ABB RobotStudio station: AutoDataCollectionRBSDone.rspag

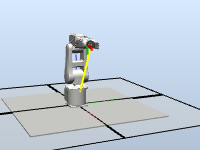
--- station ---
Station Project1 (saved by RobotStudio 6.5.7558.2005)
Controller 120-501447, task T_ROB1: task frame (RAPID world) sits at (0, 0, 10) mm in the station
Controller 120-501447
  mechanical unit ROB_1: IRB120_3_58__01, 6 joints, base frame (0, 0, 0) mm
Layout (positions relative to the parent item):
  - IRB120_3_58__01 [mechanism, from Robots\IRB120_3_58_G_01.rslib] at (0, 0, 10) mm; joint values [0, 0, 0, 0, 0, 0] (rad or m)
  - Table [part] at (-574.68, -626.92, 0) mm
  - tGripper [mechanism] at (374, 0, 640) mm, rotated rx 90 ry 0 rz 90 deg
      TCP tGripper at (14.1, 9.97, 139.57) mm
      links: ABB-TOOL-GRIPPER
  - Frame_1 [frame] at (14.1, -0.53, 139.57) mm
  - TestCyl [frame] at (160.39, -370.36, 110.04) mm
  - TestPap [frame] at (297.7, -422.52, 10) mm
  - Pointer [frame] at (82.12, -626.92, 10) mm
  - DegreeCheck1 [frame] at (285, -62, 10) mm
  - DegreeCheck2 [frame] at (285, 62, 10) mm
Attachment: IRB120_3_58__01 is attached to Table
Attachment: tGripper is attached to IRB120_3_58__01 / Link6
Collision set CollisionSet_2: Link1, Link2, Link3, Link4, Link5, Link6 against Table, near miss 0 m
Collision set CollisionSet_3: tGripper against Table, near miss 0 m

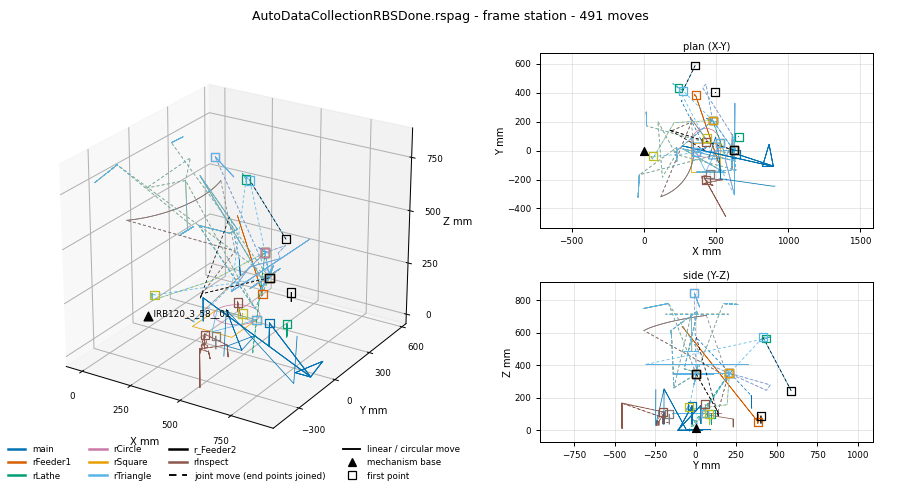
[picture p0: tool path of AutoDataCollectionRBSDone.rspag in frame station, 491 of 504 moves have a stored position in this frame; points joined in program order, loops and branches not executed]
--- Backups/120-501447/RAPID/TASK1/PROGMOD/CalibData.mod ---
MODULE CalibData
	PERS tooldata tGripper:=[TRUE,[[1.097,11.475,139.568],[0,0,0.707106781,0.707106781]],[1,[13.941,-25.105,74.149],[1,0,0,0],0,0,0]];
ENDMODULE

--- Backups/120-501447/RAPID/TASK1/PROGMOD/SERVER.mod ---
MODULE SERVER

!////////////////
!GLOBAL VARIABLES
!////////////////

!//Robot configuration
PERS tooldata currentTool := [TRUE,[[1.6,-47.2,24.1],[0.5,-0.5,-0.5,-0.5]],[1,[13.941,-25.105,74.149],[1,0,0,0],0,0,0]];
PERS wobjdata currentWobj := [FALSE,TRUE,"",[[0,0,0],[1,0,0,0]],[[0,0,0],[1,0,0,0]]];
PERS speeddata currentSpeed;
PERS zonedata currentZone;

!// Clock Synchronization
PERS bool startLog:=TRUE;
PERS bool startRob:=TRUE;

!// Mutex between logger and changing the tool and work objects
PERS bool frameMutex:=FALSE;

!//PC communication
VAR socketdev clientSocket;
VAR socketdev serverSocket;
VAR num instructionCode;
VAR num params{10};
VAR num nParams;

!PERS string ipController:= "192.168.125.1"; !robot default IP
PERS string ipController:= "127.0.0.1"; !local IP for testing in simulation
PERS num serverPort:= 5000;

!//Motion of the robot
VAR robtarget cartesianTarget;
VAR jointtarget jointsTarget;
VAR bool moveCompleted; !Set to true after finishing a Move instruction.

!//Buffered move variables
CONST num MAX_BUFFER := 512;
VAR num BUFFER_POS := 0;
VAR robtarget bufferTargets{MAX_BUFFER};
VAR speeddata bufferSpeeds{MAX_BUFFER};

!//External axis position variables
VAR extjoint externalAxis;

!//Circular move buffer
VAR robtarget circPoint;

!//Correct Instruction Execution and possible return values
VAR num ok;
CONST num SERVER_BAD_MSG :=  0;
CONST num SERVER_OK := 1;

!//Digital IO values
CONST dionum on := 1;
CONST dionum off := 0;



!////////////////
!LOCAL METHODS
!////////////////

!//Method to parse the message received from a PC
!// If correct message, loads values on:
!// - instructionCode.
!// - nParams: Number of received parameters.
!// - params{nParams}: Vector of received params.
PROC ParseMsg(string msg)
    !//Local variables
    VAR bool auxOk;
    VAR num ind:=1;
    VAR num newInd;
    VAR num length;
    VAR num indParam:=1;
    VAR string subString;
    VAR bool end := FALSE;

    !//Find the end character
    length := StrMatch(msg,1,"#");
    IF length > StrLen(msg) THEN
        !//Corrupt message
        nParams := -1;
    ELSE
        !//Read Instruction code
        newInd := StrMatch(msg,ind," ") + 1;
        subString := StrPart(msg,ind,newInd - ind - 1);
        auxOk:= StrToVal(subString, instructionCode);
        IF auxOk = FALSE THEN
            !//Impossible to read instruction code
            nParams := -1;
        ELSE
            ind := newInd;
            !//Read all instruction parameters (maximum of 8)
            WHILE end = FALSE DO
                newInd := StrMatch(msg,ind," ") + 1;
                IF newInd > length THEN
                    end := TRUE;
                ELSE
                    subString := StrPart(msg,ind,newInd - ind - 1);
                    auxOk := StrToVal(subString, params{indParam});
                    indParam := indParam + 1;
                    ind := newInd;
                ENDIF
            ENDWHILE
            nParams:= indParam - 1;
        ENDIF
    ENDIF
ENDPROC


!//Handshake between server and client:
!// - Creates socket.
!// - Waits for incoming TCP connection.
PROC ServerCreateAndConnect(string ip, num port)
    VAR string clientIP;

    SocketCreate serverSocket;
    SocketBind serverSocket, ip, port;
    SocketListen serverSocket;
    TPWrite "SERVER: Server waiting for incoming connections ...";
    WHILE SocketGetStatus(clientSocket) <> SOCKET_CONNECTED DO
        SocketAccept serverSocket,clientSocket \ClientAddress:=clientIP \Time:=WAIT_MAX;
        IF SocketGetStatus(clientSocket) <> SOCKET_CONNECTED THEN
            TPWrite "SERVER: Problem serving an incoming connection.";
            TPWrite "SERVER: Try reconnecting.";
        ENDIF
        !//Wait 0.5 seconds for the next reconnection
        WaitTime 0.5;
    ENDWHILE
    TPWrite "SERVER: Connected to IP " + clientIP;
ENDPROC


!//Parameter initialization
!// Loads default values for
!// - Tool.
!// - WorkObject.
!// - Zone.
!// - Speed.
PROC Initialize()
    currentTool := [TRUE,[[0,0,0],[1,0,0,0]],[0.001,[0,0,0.001],[1,0,0,0],0,0,0]];
    currentWobj := [FALSE,TRUE,"",[[0,0,0],[1,0,0,0]],[[0,0,0],[1,0,0,0]]];
    currentSpeed := [100, 50, 0, 0];
    currentZone := [FALSE, 0.3, 0.3,0.3,0.03,0.3,0.03]; !z0

	!Find the current external axis values so they don't move when we start
	jointsTarget := CJointT();
	externalAxis := jointsTarget.extax;
ENDPROC


!////////////////////////
!//SERVER: Main procedure
!////////////////////////
PROC main()
    !//Local variables
    VAR string receivedString;   !//Received string
    VAR string sendString;       !//Reply string
    VAR string addString;        !//String to add to the reply.
    VAR bool connected;          !//Client connected
    VAR bool reconnected;        !//Drop and reconnection happened during serving a command
    VAR robtarget cartesianPose;
    VAR jointtarget jointsPose;

    !//Motion configuration
    ConfL \Off;
    SingArea \Wrist;
    moveCompleted:= TRUE;

    !//Initialization of WorkObject, Tool, Speed and Zone
    Initialize;

    !//Socket connection
    connected:=FALSE;
    ServerCreateAndConnect ipController,serverPort;
    connected:=TRUE;

    !//Server Loop
    WHILE TRUE DO
        !//Initialization of program flow variables
        ok:=SERVER_OK;              !//Correctness of executed instruction.
        reconnected:=FALSE;         !//Has communication dropped after receiving a command?
        addString := "";

        !//Wait for a command
        SocketReceive clientSocket \Str:=receivedString \Time:=WAIT_MAX;
        ParseMsg receivedString;

        !//Execution of the command
        TEST instructionCode
            CASE 0: !Ping
                IF nParams = 0 THEN
                    ok := SERVER_OK;
                ELSE
                    ok := SERVER_BAD_MSG;
                ENDIF

            CASE 1: !Cartesian Move
                IF nParams = 7 THEN
                    cartesianTarget :=[[params{1},params{2},params{3}],
                                       [params{4},params{5},params{6},params{7}],
                                       [0,0,0,0],
                                       externalAxis];
                    ok := SERVER_OK;
                    moveCompleted := FALSE;
                    MoveL cartesianTarget, currentSpeed, currentZone, currentTool \WObj:=currentWobj ;
                    moveCompleted := TRUE;
                ELSE
                    ok := SERVER_BAD_MSG;
                ENDIF

            CASE 2: !Joint Move
                IF nParams = 6 THEN
                    jointsTarget:=[[params{1},params{2},params{3},params{4},params{5},params{6}], externalAxis];
                    ok := SERVER_OK;
                    moveCompleted := FALSE;
                    MoveAbsJ jointsTarget, currentSpeed, currentZone, currentTool \Wobj:=currentWobj;
                    moveCompleted := TRUE;
                ELSE
                    ok :=SERVER_BAD_MSG;
                ENDIF

            CASE 3: !Get Cartesian Coordinates (with current tool and workobject)
                IF nParams = 0 THEN
                    cartesianPose := CRobT(\Tool:=currentTool \WObj:=currentWObj);
                    addString := NumToStr(cartesianPose.trans.x,2) + " ";
                    addString := addString + NumToStr(cartesianPose.trans.y,2) + " ";
                    addString := addString + NumToStr(cartesianPose.trans.z,2) + " ";
                    addString := addString + NumToStr(cartesianPose.rot.q1,3) + " ";
                    addString := addString + NumToStr(cartesianPose.rot.q2,3) + " ";
                    addString := addString + NumToStr(cartesianPose.rot.q3,3) + " ";
                    addString := addString + NumToStr(cartesianPose.rot.q4,3); !End of string
                    ok := SERVER_OK;
                ELSE
                    ok :=SERVER_BAD_MSG;
                ENDIF

            CASE 4: !Get Joint Coordinates
                IF nParams = 0 THEN
                    jointsPose := CJointT();
                    addString := NumToStr(jointsPose.robax.rax_1,2) + " ";
                    addString := addString + NumToStr(jointsPose.robax.rax_2,2) + " ";
                    addString := addString + NumToStr(jointsPose.robax.rax_3,2) + " ";
                    addString := addString + NumToStr(jointsPose.robax.rax_4,2) + " ";
                    addString := addString + NumToStr(jointsPose.robax.rax_5,2) + " ";
                    addString := addString + NumToStr(jointsPose.robax.rax_6,2); !End of string
                    ok := SERVER_OK;
                ELSE
                    ok:=SERVER_BAD_MSG;
                ENDIF
			CASE 5: !Get external axis positions
                IF nParams = 0 THEN
                    jointsPose := CJointT();
                    addString := StrPart(NumToStr(jointsTarget.extax.eax_a, 2),1,8) + " ";
                    addString := addString + StrPart(NumToStr(jointsTarget.extax.eax_b,2),1,8) + " ";
                    addString := addString + StrPart(NumToStr(jointsTarget.extax.eax_c,2),1,8) + " ";
                    addString := addString + StrPart(NumToStr(jointsTarget.extax.eax_d,2),1,8) + " ";
                    addString := addString + StrPart(NumToStr(jointsTarget.extax.eax_e,2),1,8) + " ";
                    addString := addString + StrPart(NumToStr(jointsTarget.extax.eax_f,2),1,8); !End of string
                    ok := SERVER_OK;
                ELSE
                    ok:=SERVER_BAD_MSG;
                ENDIF

            CASE 6: !Set Tool
                IF nParams = 7 THEN
		   WHILE (frameMutex) DO
		        WaitTime .01; !// If the frame is being used by logger, wait here
		   ENDWHILE
		frameMutex:= TRUE;
                    currentTool.tframe.trans.x:=params{1};
                    currentTool.tframe.trans.y:=params{2};
                    currentTool.tframe.trans.z:=params{3};
                    currentTool.tframe.rot.q1:=params{4};
                    currentTool.tframe.rot.q2:=params{5};
                    currentTool.tframe.rot.q3:=params{6};
                    currentTool.tframe.rot.q4:=params{7};
                    ok := SERVER_OK;
		    frameMutex:= FALSE;
                ELSE
                    ok:=SERVER_BAD_MSG;
                ENDIF

            CASE 7: !Set Work Object
                IF nParams = 7 THEN
                    currentWobj.oframe.trans.x:=params{1};
                    currentWobj.oframe.trans.y:=params{2};
                    currentWobj.oframe.trans.z:=params{3};
                    currentWobj.oframe.rot.q1:=params{4};
                    currentWobj.oframe.rot.q2:=params{5};
                    currentWobj.oframe.rot.q3:=params{6};
                    currentWobj.oframe.rot.q4:=params{7};
                    ok := SERVER_OK;
                ELSE
                    ok:=SERVER_BAD_MSG;
                ENDIF

            CASE 8: !Set Speed of the Robot
                IF nParams = 4 THEN
                    currentSpeed.v_tcp:=params{1};
                    currentSpeed.v_ori:=params{2};
                    currentSpeed.v_leax:=params{3};
                    currentSpeed.v_reax:=params{4};
                    ok := SERVER_OK;
                ELSEIF nParams = 2 THEN
					currentSpeed.v_tcp:=params{1};
					currentSpeed.v_ori:=params{2};
					ok := SERVER_OK;
				ELSE
                    ok:=SERVER_BAD_MSG;
                ENDIF

            CASE 9: !Set zone data
                IF nParams = 4 THEN
                    IF params{1}=1 THEN
                        currentZone.finep := TRUE;
                        currentZone.pzone_tcp := 0.0;
                        currentZone.pzone_ori := 0.0;
                        currentZone.zone_ori := 0.0;
                    ELSE
                        currentZone.finep := FALSE;
                        currentZone.pzone_tcp := params{2};
                        currentZone.pzone_ori := params{3};
                        currentZone.zone_ori := params{4};
                    ENDIF
                    ok := SERVER_OK;
                ELSE
                    ok:=SERVER_BAD_MSG;
                ENDIF

            CASE 30: !Add Cartesian Coordinates to buffer
                IF nParams = 7 THEN
                    cartesianTarget :=[[params{1},params{2},params{3}],
                                        [params{4},params{5},params{6},params{7}],
                                        [0,0,0,0],
                                        externalAxis];
                    IF BUFFER_POS < MAX_BUFFER THEN
                        BUFFER_POS := BUFFER_POS + 1;
                        bufferTargets{BUFFER_POS} := cartesianTarget;
                        bufferSpeeds{BUFFER_POS} := currentSpeed;
                    ENDIF
                    ok := SERVER_OK;
                ELSE
                    ok:=SERVER_BAD_MSG;
                ENDIF

            CASE 31: !Clear Cartesian Buffer
                IF nParams = 0 THEN
                    BUFFER_POS := 0;
                    ok := SERVER_OK;
                ELSE
                    ok:=SERVER_BAD_MSG;
                ENDIF

            CASE 32: !Get Buffer Size)
                IF nParams = 0 THEN
                    addString := NumToStr(BUFFER_POS,2);
                    ok := SERVER_OK;
                ELSE
                    ok:=SERVER_BAD_MSG;
                ENDIF

            CASE 33: !Execute moves in cartesianBuffer as linear moves
                IF nParams = 0 THEN
                    FOR i FROM 1 TO (BUFFER_POS) DO
                        MoveL bufferTargets{i}, bufferSpeeds{i}, currentZone, currentTool \WObj:=currentWobj ;
                    ENDFOR
                    ok := SERVER_OK;
                ELSE
                    ok:=SERVER_BAD_MSG;
                ENDIF

            CASE 34: !External Axis move
                IF nParams = 6 THEN
                    externalAxis :=[params{1},params{2},params{3},params{4},params{5},params{6}];
                    jointsTarget := CJointT();
                    jointsTarget.extax := externalAxis;
                    ok := SERVER_OK;
                    moveCompleted := FALSE;
                    MoveAbsJ jointsTarget, currentSpeed, currentZone, currentTool \Wobj:=currentWobj;
                    moveCompleted := TRUE;
                ELSE
                    ok :=SERVER_BAD_MSG;
                ENDIF

            CASE 35: !Specify circPoint for circular move, and then wait on toPoint
                IF nParams = 7 THEN
                    circPoint :=[[params{1},params{2},params{3}],
                                [params{4},params{5},params{6},params{7}],
                                [0,0,0,0],
                                externalAxis];
                    ok := SERVER_OK;
                ELSE
                    ok:=SERVER_BAD_MSG;
                ENDIF

            CASE 36: !specify toPoint, and use circPoint specified previously
                IF nParams = 7 THEN
                    cartesianTarget :=[[params{1},params{2},params{3}],
                                        [params{4},params{5},params{6},params{7}],
                                        [0,0,0,0],
                                        externalAxis];
                    MoveC circPoint, cartesianTarget, currentSpeed, currentZone, currentTool \WObj:=currentWobj ;
                    ok := SERVER_OK;
                ELSE
                    ok:=SERVER_BAD_MSG;
                ENDIF

            CASE 37: !Sets doGrip to input value
                IF nParams = 1 THEN
                    SetDo doGrip, params{1};
                    ok := SERVER_OK;
                ELSE
                    ok:=SERVER_BAD_MSG;
                ENDIF

            CASE 38: !Sets doVacume to input value
                IF nParams = 1 THEN
                    SetDo doVacume, params{1};
                    ok := SERVER_OK;
                ELSE
                    ok:=SERVER_BAD_MSG;
                ENDIF

            CASE 39: !Sets doTrace to input value
                IF nParams = 1 THEN
                    SetDo doTrace, params{1};
                    ok := SERVER_OK;
                ELSE
                    ok:=SERVER_BAD_MSG;
                ENDIF

            CASE 41: !Set Advanced Tool
                IF nParams = 8 THEN
		   WHILE (frameMutex) DO
		        WaitTime .01; !// If the frame is being used by logger, wait here
		   ENDWHILE
		frameMutex:= TRUE;
                    currentTool.tload.mass:=params{1};
                    currentTool.tload.cog.x:=params{2};
                    currentTool.tload.cog.y:=params{3};
                    currentTool.tload.cog.z:=params{4};
                    currentTool.tload.aom.q1:=params{5};
                    currentTool.tload.aom.q2:=params{6};
                    currentTool.tload.aom.q3:=params{7};
                    currentTool.tload.aom.q4:=params{8};
                    ok := SERVER_OK;
		    frameMutex:= FALSE;
                ELSE
                    ok:=SERVER_BAD_MSG;
                ENDIF

            CASE 98: !returns current robot info: serial number, robotware version, and robot type
                IF nParams = 0 THEN
                    addString := GetSysInfo(\SerialNo) + "*";
                    addString := addString + GetSysInfo(\SWVersion) + "*";
                    addString := addString + GetSysInfo(\RobotType);
                    ok := SERVER_OK;
                ELSE
                    ok :=SERVER_BAD_MSG;
                ENDIF

            CASE 99: !Close Connection
                IF nParams = 0 THEN
                    TPWrite "SERVER: Client has closed connection.";
                    connected := FALSE;
                    !//Closing the server
                    SocketClose clientSocket;
                    SocketClose serverSocket;

                    !Reinitiate the server
                    ServerCreateAndConnect ipController,serverPort;
                    connected := TRUE;
                    reconnected := TRUE;
                    ok := SERVER_OK;
                ELSE
                    ok := SERVER_BAD_MSG;
                ENDIF
            DEFAULT:
                TPWrite "SERVER: Illegal instruction code";
                ok := SERVER_BAD_MSG;
        ENDTEST

        !Compose the acknowledge string to send back to the client
        IF connected = TRUE THEN
            IF reconnected = FALSE THEN
			    IF SocketGetStatus(clientSocket) = SOCKET_CONNECTED THEN
				    sendString := NumToStr(instructionCode,0);
                    sendString := sendString + " " + NumToStr(ok,0);
                    sendString := sendString + " " + addString;
                    SocketSend clientSocket \Str:=sendString;
			    ENDIF
            ENDIF
        ENDIF
    ENDWHILE

ERROR (LONG_JMP_ALL_ERR)
    TPWrite "SERVER: ------";
    TPWrite "SERVER: Error Handler:" + NumtoStr(ERRNO,0);
    TEST ERRNO
        CASE ERR_SOCK_CLOSED:
            TPWrite "SERVER: Lost connection to the client.";
            TPWrite "SERVER: Closing socket and restarting.";
            TPWrite "SERVER: ------";
            connected:=FALSE;
            !//Closing the server
            SocketClose clientSocket;
            SocketClose serverSocket;
            !//Reinitiate the server
            ServerCreateAndConnect ipController,serverPort;
            reconnected:= FALSE;
            connected:= TRUE;
            RETRY;
        DEFAULT:
            TPWrite "SERVER: Unknown error.";
            TPWrite "SERVER: Closing socket and restarting.";
            TPWrite "SERVER: ------";
            connected:=FALSE;
            !//Closing the server
            SocketClose clientSocket;
            SocketClose serverSocket;
            !//Reinitiate the server
            ServerCreateAndConnect ipController,serverPort;
            reconnected:= FALSE;
            connected:= TRUE;
            RETRY;
    ENDTEST
ENDPROC

ENDMODULE

--- Backups/120-501447/RAPID/TASK1/SYSMOD/SysTools.sys ---
MODULE SysTools(SYSMODULE)
    CONST jointtarget jZeroJoint:=[[0.489285,0.00104285,0.00208998,0.00446524,-0.00462914,-0.00385281],[9E+09,9E+09,9E+09,9E+09,9E+09,9E+09]];

    PROC jZero()
		MoveAbsJ jZeroJoint\NoEOffs, v1000, z50, tool0;
	ENDPROC
ENDMODULE

--- Backups/120-501447/RAPID/TASK2/PROGMOD/LOGGER.mod ---
MODULE LOGGER

!////////////////
!GLOBAL VARIABLES
!////////////////
!PC communication
VAR socketdev clientSocket;
VAR socketdev serverSocket;
PERS string ipController;
PERS num loggerPort:= 5001;

!Robot configuration
PERS tooldata currentTool;
PERS wobjdata currentWobj;
VAR speeddata currentSpeed;
VAR zonedata currentZone;

!//Logger sampling rate
!PERS num loggerWaitTime:= 0.01;  !Recommended for real controller
PERS num loggerWaitTime:= 0.1;    !Recommended for virtual controller

PROC ServerCreateAndConnect(string ip, num port)
	VAR string clientIP;

	SocketCreate serverSocket;
	SocketBind serverSocket, ip, port;
	SocketListen serverSocket;
	TPWrite "LOGGER: Logger waiting for incomming connections ...";
	WHILE SocketGetStatus(clientSocket) <> SOCKET_CONNECTED DO
		SocketAccept serverSocket,clientSocket \ClientAddress:=clientIP \Time:=WAIT_MAX;
		IF SocketGetStatus(clientSocket) <> SOCKET_CONNECTED THEN
			TPWrite "LOGGER: Problem serving an incomming connection.";
			TPWrite "LOGGER: Try reconnecting.";
		ENDIF
		 !Wait 0.5 seconds for the next reconnection
		 WaitTime 0.5;
	ENDWHILE
	TPWrite "LOGGER: Connected to IP " + clientIP;
ENDPROC

PROC main()
	VAR string data;
	VAR robtarget position;
	VAR jointtarget joints;
    VAR string sendString;
	VAR bool connected;

	VAR string date;
	VAR string time;
	VAR clock timer;

	date:= CDate();
	time:= CTime();
    ClkStart timer;

	connected:=FALSE;
	ServerCreateAndConnect ipController,loggerPort;
	connected:=TRUE;
	WHILE TRUE DO

		!Cartesian Coordinates
		position := CRobT(\Tool:=currentTool \WObj:=currentWObj);
		data := "# 0 ";
		data := data + date + " " + time + " ";
		data := data + NumToStr(ClkRead(timer),2) + " ";
		data := data + NumToStr(position.trans.x,1) + " ";
		data := data + NumToStr(position.trans.y,1) + " ";
		data := data + NumToStr(position.trans.z,1) + " ";
		data := data + NumToStr(position.rot.q1,3) + " ";
		data := data + NumToStr(position.rot.q2,3) + " ";
		data := data + NumToStr(position.rot.q3,3) + " ";
		data := data + NumToStr(position.rot.q4,3); !End of string
		IF connected = TRUE THEN
			SocketSend clientSocket \Str:=data;
		ENDIF
		WaitTime loggerWaitTime;

		!Joint Coordinates
		joints := CJointT();
		data := "# 1 ";
		data := data + date + " " + time + " ";
		data := data + NumToStr(ClkRead(timer),2) + " ";
		data := data + NumToStr(joints.robax.rax_1,2) + " ";
		data := data + NumToStr(joints.robax.rax_2,2) + " ";
		data := data + NumToStr(joints.robax.rax_3,2) + " ";
		data := data + NumToStr(joints.robax.rax_4,2) + " ";
		data := data + NumToStr(joints.robax.rax_5,2) + " ";
		data := data + NumToStr(joints.robax.rax_6,2); !End of string
		IF connected = TRUE THEN
			SocketSend clientSocket \Str:=data;
		ENDIF
		WaitTime loggerWaitTime;
	ENDWHILE
	ERROR
	IF ERRNO=ERR_SOCK_CLOSED THEN
		TPWrite "LOGGER: Client has closed connection.";
	ELSE
		TPWrite "LOGGER: Connection lost: Unknown problem.";
	ENDIF
	connected:=FALSE;
	!Closing the server
	SocketClose clientSocket;
	SocketClose serverSocket;
	!Reinitiate the server
	ServerCreateAndConnect ipController,loggerPort;
	connected:= TRUE;
	RETRY;
ENDPROC

ENDMODULE

--- Backups/120-501447/HOME/Conveyor/MainModule.mod ---
MODULE MainModule
	TASK PERS tooldata tPen:=[TRUE,[[0.147757,-83.6911,144.451],[0.738156,0.674482,-0.0103991,-0.00950206]],[0.8,[1.7,0,108.7],[1,0,0,0],0.011,0.006,0.009]];
	CONST robtarget p30:=[[469.22,99.75,8.79],[0.0216335,0.64282,0.765703,-0.00355185],[0,0,0,1],[9E+09,9E+09,9E+09,9E+09,9E+09,9E+09]];
	CONST robtarget pstart:=[[512.08,-48.21,10.23],[0.0215519,0.642623,0.765869,-0.00379738],[-1,-1,0,1],[9E+09,9E+09,9E+09,9E+09,9E+09,9E+09]];
	CONST robtarget p10:=[[268.52,32.55,142.20],[0.0387242,0.836099,0.54718,0.00566096],[0,0,0,1],[9E+09,9E+09,9E+09,9E+09,9E+09,9E+09]];
	CONST robtarget p20:=[[268.52,32.55,29.70],[0.0387219,0.8361,0.547177,0.00566567],[0,0,0,1],[9E+09,9E+09,9E+09,9E+09,9E+09,9E+09]];
	CONST robtarget p40:=[[505.98,113.33,4.46],[0.0367854,0.831559,0.554195,0.00482753],[0,0,0,1],[9E+09,9E+09,9E+09,9E+09,9E+09,9E+09]];
	CONST robtarget p50:=[[461.62,115.15,-8.30],[0.0367965,0.831555,0.5542,0.00481934],[0,0,0,1],[9E+09,9E+09,9E+09,9E+09,9E+09,9E+09]];
	CONST robtarget p60:=[[525.97,169.03,3.52],[0.0368121,0.8315,0.554282,0.00472824],[0,0,0,1],[9E+09,9E+09,9E+09,9E+09,9E+09,9E+09]];
	CONST robtarget p70:=[[597.29,115.27,0.65],[0.0368322,0.831492,0.554294,0.00471092],[0,0,0,1],[9E+09,9E+09,9E+09,9E+09,9E+09,9E+09]];
	CONST robtarget p80:=[[569.04,115.26,0.68],[0.036874,0.831516,0.554254,0.00474228],[0,0,0,1],[9E+09,9E+09,9E+09,9E+09,9E+09,9E+09]];
	CONST robtarget p90:=[[579.87,-35.31,-1.57],[0.0368611,0.831471,0.554322,0.00471824],[0,0,0,1],[9E+09,9E+09,9E+09,9E+09,9E+09,9E+09]];
	CONST robtarget p100:=[[547.53,-9.26,-1.58],[0.0368624,0.831474,0.554318,0.00469294],[0,0,0,1],[9E+09,9E+09,9E+09,9E+09,9E+09,9E+09]];
	CONST robtarget p110:=[[532.30,-194.48,243.92],[0.0367212,0.831611,0.55412,0.00498134],[-1,0,0,1],[9E+09,9E+09,9E+09,9E+09,9E+09,9E+09]];
	TASK PERS wobjdata wFixture1:=[FALSE,TRUE,"",[[0,0,0],[1,0,0,0]],[[357.689,-176.134,-17.7192],[0.999991,-0.00111829,0.000705852,-0.00392021]]];
	TASK PERS wobjdata wobj1:=[FALSE,TRUE,"",[[0,0,0],[1,0,0,0]],[[372.049,-59.0817,-2.31291],[0.999964,0.00101619,0.00195787,0.00815211]]];
	CONST robtarget pOverPart:=[[-6.04,442.92,43.54],[0.0169854,0.295249,0.953564,0.0570485],[0,-1,1,1],[9E+09,9E+09,9E+09,9E+09,9E+09,9E+09]];
	CONST robtarget pOnPart:=[[143.48,-25.45,633.13],[0.527232,0.474806,0.509036,-0.487305],[0,-1,-1,1],[9E+09,9E+09,9E+09,9E+09,9E+09,9E+09]];
	PROC main()
		MoveJ p10, v1000, z50, tPen\WObj:=wobj1;
		MoveL p20, v1000, fine, tPen\WObj:=wobj1;
		Set doGrip;
		MoveL p10, v1000, fine, tPen\WObj:=wobj1;
		MoveL [[523.80,-56.63,-8.74],[0.0367413,0.831596,0.554142,0.00493633],[0,0,0,1],[9E+09,9E+09,9E+09,9E+09,9E+09,9E+09]], v1000, fine, tPen\WObj:=wobj1;
		MoveL [[449.04,-57.95,-7.57],[0.0367587,0.831587,0.554155,0.00488328],[0,0,1,1],[9E+09,9E+09,9E+09,9E+09,9E+09,9E+09]], v1000, fine, tPen\WObj:=wobj1;
		MoveL [[497.17,94.80,-7.58],[0.0367718,0.831577,0.554169,0.00486949],[0,0,0,1],[9E+09,9E+09,9E+09,9E+09,9E+09,9E+09]], v1000, fine, tPen\WObj:=wobj1;
		MoveL [[524.39,-59.04,-6.34],[0.037286,0.83168,0.553975,0.00527583],[0,0,0,1],[9E+09,9E+09,9E+09,9E+09,9E+09,9E+09]], v1000, fine, tPen\WObj:=wobj1;
		MoveL p10, v1000, fine, tPen;
		MoveL p20, v1000, fine, tPen;
		Reset doGrip;
	ENDPROC
	PROC rGotoCal()
		MoveAbsJ jposCal\NoEOffs, v1000, z50, tPen\WObj:=wobj1;
	ENDPROC
	PROC rFeeder1()
		MoveJ pOverPart, v500, z30, tPen\WObj:=wobj1;
		MoveL pOnPart, v500, fine, tPen\WObj:=wobj1;
		Set doGrip;
		MoveL pOverPart, v500, z30, tPen\WObj:=wobj1;
		RETURN;
	ENDPROC
ENDMODULE

--- Backups/120-501447/HOME/Conveyor/TCPZ_tPen.mod ---
MODULE TCPZ_tPen
	! Points are read in order of declaration.
  ! Please do not change the order of points!

  LOCAL PERS robtarget pTCPZ_Point1:=[[382.153,36.8026,340.3493],[0.538514792919159,0.222296640276909,0.790146291255951,0.190406858921051],[0,0,0,1],[9E+09,9E+09,9E+09,9E+09,9E+09,9E+09]];
	LOCAL PERS robtarget pTCPZ_Point2:=[[383.4106,-54.66603,352.9551],[0.307397365570068,0.748442351818085,0.310303926467896,0.499051481485367],[-1,0,1,1],[9E+09,9E+09,9E+09,9E+09,9E+09,9E+09]];
	LOCAL PERS robtarget pTCPZ_Point3:=[[340.256,-13.576,241.934],[0.634813845157623,0.35798105597496,0.338523089885712,0.595200002193451],[-1,0,0,1],[9E+09,9E+09,9E+09,9E+09,9E+09,9E+09]];
	LOCAL PERS robtarget pTCPZ_Point4:=[[371.1446,-16.74413,343.3362],[0.484932452440262,0.54239946603775,0.505667269229889,0.463620454072952],[-1,0,1,1],[9E+09,9E+09,9E+09,9E+09,9E+09,9E+09]];
	LOCAL PERS robtarget pTCPZ_ElongZ:=[[365.5099,-16.1815,420.0958],[0.503183424472809,0.523792386054993,0.483616411685944,0.488429248332977],[-1,0,1,1],[9E+09,9E+09,9E+09,9E+09,9E+09,9E+09]];

ENDMODULE

--- Backups/120-501447/HOME/Conveyor/Wobj_wFixture1.mod ---
MODULE Wobj_wFixture1
	! Points are read in order of declaration.
  ! Please do not change the order of points!

  LOCAL PERS robtarget pWobj_O_PointX1:=[[375.484,-176.2736,-17.74421],[0.00141646177507937,-0.64477950334549,-0.764364421367645,-0.00174713658634573],[-1,-1,0,1],[9E+09,9E+09,9E+09,9E+09,9E+09,9E+09]];
	LOCAL PERS robtarget pWobj_O_PointX2:=[[689.4256,-178.7356,-18.18466],[0.00207201461307704,-0.646406650543213,-0.762987077236176,-0.00188234634697437],[-1,-1,1,1],[9E+09,9E+09,9E+09,9E+09,9E+09,9E+09]];
	LOCAL PERS robtarget pWobj_O_PointY1:=[[361.8714,357.4471,-18.91562],[0.00154154072515666,-0.644824087619781,-0.764327049255371,-0.00151761737652123],[0,0,0,1],[9E+09,9E+09,9E+09,9E+09,9E+09,9E+09]];
	CONST jointtarget jposCal:=[[0.0258162,-0.0104883,-0.0155317,-0.00860849,-0.0253093,-0.00857693],[9E+09,9E+09,9E+09,9E+09,9E+09,9E+09]];

ENDMODULE

--- Backups/120-501447/HOME/Conveyor/Wobj_wobj1.mod ---
MODULE Wobj_wobj1
	! Points are read in order of declaration.
  ! Please do not change the order of points!

  LOCAL PERS robtarget pWobj_O_PointX1:=[[373.4612,-59.05866,-2.318419],[0.0375104658305645,0.834795832633972,0.549128353595734,-0.012865555472672],[0,0,1,1],[9E+09,9E+09,9E+09,9E+09,9E+09,9E+09]];
	LOCAL PERS robtarget pWobj_O_PointX2:=[[701.291,-53.71179,-3.59682],[0.0375093184411526,0.834785938262939,0.54914253950119,-0.0129095437005162],[0,0,0,1],[9E+09,9E+09,9E+09,9E+09,9E+09,9E+09]];
	LOCAL PERS robtarget pWobj_O_PointY1:=[[364.21,421.8124,-1.320101],[0.0375351272523403,0.83477908372879,0.549150884151459,-0.012924118898809],[0,1,0,1],[9E+09,9E+09,9E+09,9E+09,9E+09,9E+09]];

ENDMODULE

--- Backups/120-501447/HOME/Conveyor/Conveyor/MainModule.mod ---
MODULE MainModule
	TASK PERS tooldata tPen:=[TRUE,[[0.147757,-83.6911,144.451],[0.738156,0.674482,-0.0103991,-0.00950206]],[0.8,[1.7,0,108.7],[1,0,0,0],0.011,0.006,0.009]];
	CONST robtarget p30:=[[469.22,99.75,8.79],[0.0216335,0.64282,0.765703,-0.00355185],[0,0,0,1],[9E+09,9E+09,9E+09,9E+09,9E+09,9E+09]];
	CONST robtarget pstart:=[[512.08,-48.21,10.23],[0.0215519,0.642623,0.765869,-0.00379738],[-1,-1,0,1],[9E+09,9E+09,9E+09,9E+09,9E+09,9E+09]];
	CONST robtarget p10:=[[268.52,32.55,142.20],[0.0387242,0.836099,0.54718,0.00566096],[0,0,0,1],[9E+09,9E+09,9E+09,9E+09,9E+09,9E+09]];
	CONST robtarget p20:=[[268.52,32.55,29.70],[0.0387219,0.8361,0.547177,0.00566567],[0,0,0,1],[9E+09,9E+09,9E+09,9E+09,9E+09,9E+09]];
	CONST robtarget p40:=[[505.98,113.33,4.46],[0.0367854,0.831559,0.554195,0.00482753],[0,0,0,1],[9E+09,9E+09,9E+09,9E+09,9E+09,9E+09]];
	CONST robtarget p50:=[[461.62,115.15,-8.30],[0.0367965,0.831555,0.5542,0.00481934],[0,0,0,1],[9E+09,9E+09,9E+09,9E+09,9E+09,9E+09]];
	CONST robtarget p60:=[[525.97,169.03,3.52],[0.0368121,0.8315,0.554282,0.00472824],[0,0,0,1],[9E+09,9E+09,9E+09,9E+09,9E+09,9E+09]];
	CONST robtarget p70:=[[597.29,115.27,0.65],[0.0368322,0.831492,0.554294,0.00471092],[0,0,0,1],[9E+09,9E+09,9E+09,9E+09,9E+09,9E+09]];
	CONST robtarget p80:=[[569.04,115.26,0.68],[0.036874,0.831516,0.554254,0.00474228],[0,0,0,1],[9E+09,9E+09,9E+09,9E+09,9E+09,9E+09]];
	CONST robtarget p90:=[[579.87,-35.31,-1.57],[0.0368611,0.831471,0.554322,0.00471824],[0,0,0,1],[9E+09,9E+09,9E+09,9E+09,9E+09,9E+09]];
	CONST robtarget p100:=[[547.53,-9.26,-1.58],[0.0368624,0.831474,0.554318,0.00469294],[0,0,0,1],[9E+09,9E+09,9E+09,9E+09,9E+09,9E+09]];
	CONST robtarget p110:=[[532.30,-194.48,243.92],[0.0367212,0.831611,0.55412,0.00498134],[-1,0,0,1],[9E+09,9E+09,9E+09,9E+09,9E+09,9E+09]];
	TASK PERS wobjdata wFixture1:=[FALSE,TRUE,"",[[0,0,0],[1,0,0,0]],[[357.689,-176.134,-17.7192],[0.999991,-0.00111829,0.000705852,-0.00392021]]];
	TASK PERS wobjdata wobj1:=[FALSE,TRUE,"",[[0,0,0],[1,0,0,0]],[[372.049,-59.0817,-2.31291],[0.999964,0.00101619,0.00195787,0.00815211]]];
	CONST robtarget pOverPart:=[[-12.15,445.19,84.22],[0.0344175,0.27264,0.961398,0.0139876],[0,-1,1,1],[9E+09,9E+09,9E+09,9E+09,9E+09,9E+09]];
	CONST robtarget pOnPart:=[[-10.40,443.03,33.34],[0.0408588,0.27536,0.960135,0.0254239],[0,-1,0,1],[9E+09,9E+09,9E+09,9E+09,9E+09,9E+09]];
	PROC main()
		MoveJ p10, v1000, z50, tPen\WObj:=wobj1;
		MoveL p20, v1000, fine, tPen\WObj:=wobj1;
		Set doGrip;
		MoveL p10, v1000, fine, tPen\WObj:=wobj1;
		MoveL [[523.80,-56.63,-8.74],[0.0367413,0.831596,0.554142,0.00493633],[0,0,0,1],[9E+09,9E+09,9E+09,9E+09,9E+09,9E+09]], v1000, fine, tPen\WObj:=wobj1;
		MoveL [[449.04,-57.95,-7.57],[0.0367587,0.831587,0.554155,0.00488328],[0,0,1,1],[9E+09,9E+09,9E+09,9E+09,9E+09,9E+09]], v1000, fine, tPen\WObj:=wobj1;
		MoveL [[497.17,94.80,-7.58],[0.0367718,0.831577,0.554169,0.00486949],[0,0,0,1],[9E+09,9E+09,9E+09,9E+09,9E+09,9E+09]], v1000, fine, tPen\WObj:=wobj1;
		MoveL [[524.39,-59.04,-6.34],[0.037286,0.83168,0.553975,0.00527583],[0,0,0,1],[9E+09,9E+09,9E+09,9E+09,9E+09,9E+09]], v1000, fine, tPen\WObj:=wobj1;
		MoveL p10, v1000, fine, tPen;
		MoveL p20, v1000, fine, tPen;
		Reset doGrip;
	ENDPROC
	PROC rGotoCal()
		MoveAbsJ jposCal\NoEOffs, v1000, z50, tPen\WObj:=wobj1;
	ENDPROC
	PROC rFeeder1()
		MoveJ pOverPart, v500, z30, tPen\WObj:=wobj1;
		MoveL pOnPart, v500, fine, tPen\WObj:=wobj1;
		Set doGrip;
		MoveL pOverPart, v500, z30, tPen\WObj:=wobj1;
		RETURN;
	ENDPROC
	PROC rLathe()
		CONST robtarget pOverLathe:=[[286.75,151.65,90.52],[0.0344064,0.272705,0.961381,0.0139323],[-1,-1,1,1],[9E+09,9E+09,9E+09,9E+09,9E+09,9E+09]];
		CONST robtarget pInLathe:=[[287.00,151.52,27.63],[0.0344156,0.2727,0.961382,0.0139384],[-1,-1,1,1],[9E+09,9E+09,9E+09,9E+09,9E+09,9E+09]];
		MoveJ pOverLathe, v500, z10, tPen\WObj:=wobj1;
		MoveL pInLathe, v500, fine, tPen\WObj:=wobj1;
		Reset doGrip;
		MoveL pOverLathe, v500, fine, tPen\WObj:=wobj1;
	ENDPROC
ENDMODULE

--- Backups/120-501447/HOME/Conveyor/Conveyor/Circle/MainModule.mod ---
MODULE MainModule
	CONST robtarget pHome:=[[429.22,11.33,552.83],[0.320322,0.339193,0.846628,0.256051],[-1,-2,2,1],[9E+09,9E+09,9E+09,9E+09,9E+09,9E+09]];
	CONST robtarget pBegin:=[[528.66,54.57,92.32],[0.252253,0.281148,0.656612,0.652828],[0,-1,1,1],[9E+09,9E+09,9E+09,9E+09,9E+09,9E+09]];
	CONST robtarget pGrab:=[[264.31,346.00,124.68],[0.239865,0.287491,0.669033,0.642034],[0,0,1,1],[9E+09,9E+09,9E+09,9E+09,9E+09,9E+09]];
	CONST robtarget pStart:=[[260.93,343.33,202.12],[0.252283,0.28114,0.656668,0.652764],[0,0,0,1],[9E+09,9E+09,9E+09,9E+09,9E+09,9E+09]];
	VAR num nFkey:=0;
    PROC main()

		TPErase;
		TPReadFK nFKey, "Choose", "CIRCLE", "SQUARE", "TRIANGLE", stEmpty, stEmpty;
		TEST nFkey

        CASE 1:
            rCircle;
        CASE 2:
            rSquare;
        CASE 3:
            rTriangle;
        DEFAULT:
        ENDTEST
        MoveJ pHome, v1000, z50, tool0;
		MoveJ pStart, v1000, z50, tool0;
		MoveL pGrab, v1000, fine, tool0;
		Set doGrip;
		MoveL pStart, v1000, fine, tool0;
	ENDPROC
    PROC rCircle()
		MoveL pBegin, v500, fine, tool0;
		MoveC Offs(pBegin,-100,-100,0), Offs(pBegin,-200,0,0), v500, z1, tool0;
		MoveC Offs(pBegin,-100,100,0), pBegin, v500, z1, tool0;
    ENDPROC
	PROC rSquare()
		MoveL pBegin, v1000, z50, tool0;
		MoveL Offs(pBegin,-200,0,0), v1000, z0, tool0;
		MoveL Offs(pBegin,-200,-200,0), v1000, z0, tool0;
		MoveL Offs(pBegin,0,-200,0), v1000, z0, tool0;
		MoveL pBegin, v1000, z50, tool0;
	ENDPROC
	PROC rTriangle()
		MoveL pBegin, v1000, z50, tool0;
		MoveL Offs(pBegin,-100,-200,0), v1000, z0, tool0;
		MoveL Offs(pBegin,-200,0,0), v1000, z0, tool0;
		MoveL pBegin, v1000, z50, tool0;
	ENDPROC
ENDMODULE

--- Backups/120-501447/HOME/Conveyor/Conveyor/Lathe/MainModule.mod ---
MODULE MainModule
	TASK PERS tooldata tPen:=[TRUE,[[0.147757,-83.6911,144.451],[0.738156,0.674482,-0.0103991,-0.00950206]],[0.8,[1.7,0,108.7],[1,0,0,0],0.011,0.006,0.009]];
	CONST robtarget p30:=[[469.22,99.75,8.79],[0.0216335,0.64282,0.765703,-0.00355185],[0,0,0,1],[9E+09,9E+09,9E+09,9E+09,9E+09,9E+09]];
	CONST robtarget pstart:=[[512.08,-48.21,10.23],[0.0215519,0.642623,0.765869,-0.00379738],[-1,-1,0,1],[9E+09,9E+09,9E+09,9E+09,9E+09,9E+09]];
	CONST robtarget p10:=[[268.52,32.55,142.20],[0.0387242,0.836099,0.54718,0.00566096],[0,0,0,1],[9E+09,9E+09,9E+09,9E+09,9E+09,9E+09]];
	CONST robtarget p20:=[[268.52,32.55,29.70],[0.0387219,0.8361,0.547177,0.00566567],[0,0,0,1],[9E+09,9E+09,9E+09,9E+09,9E+09,9E+09]];
	CONST robtarget p40:=[[505.98,113.33,4.46],[0.0367854,0.831559,0.554195,0.00482753],[0,0,0,1],[9E+09,9E+09,9E+09,9E+09,9E+09,9E+09]];
	CONST robtarget p50:=[[461.62,115.15,-8.30],[0.0367965,0.831555,0.5542,0.00481934],[0,0,0,1],[9E+09,9E+09,9E+09,9E+09,9E+09,9E+09]];
	CONST robtarget p60:=[[525.97,169.03,3.52],[0.0368121,0.8315,0.554282,0.00472824],[0,0,0,1],[9E+09,9E+09,9E+09,9E+09,9E+09,9E+09]];
	CONST robtarget p70:=[[597.29,115.27,0.65],[0.0368322,0.831492,0.554294,0.00471092],[0,0,0,1],[9E+09,9E+09,9E+09,9E+09,9E+09,9E+09]];
	CONST robtarget p80:=[[569.04,115.26,0.68],[0.036874,0.831516,0.554254,0.00474228],[0,0,0,1],[9E+09,9E+09,9E+09,9E+09,9E+09,9E+09]];
	CONST robtarget p90:=[[579.87,-35.31,-1.57],[0.0368611,0.831471,0.554322,0.00471824],[0,0,0,1],[9E+09,9E+09,9E+09,9E+09,9E+09,9E+09]];
	CONST robtarget p100:=[[547.53,-9.26,-1.58],[0.0368624,0.831474,0.554318,0.00469294],[0,0,0,1],[9E+09,9E+09,9E+09,9E+09,9E+09,9E+09]];
	CONST robtarget p110:=[[532.30,-194.48,243.92],[0.0367212,0.831611,0.55412,0.00498134],[-1,0,0,1],[9E+09,9E+09,9E+09,9E+09,9E+09,9E+09]];
	TASK PERS wobjdata wFixture1:=[FALSE,TRUE,"",[[0,0,0],[1,0,0,0]],[[357.689,-176.134,-17.7192],[0.999991,-0.00111829,0.000705852,-0.00392021]]];
	TASK PERS wobjdata wobj1:=[FALSE,TRUE,"",[[0,0,0],[1,0,0,0]],[[372.049,-59.0817,-2.31291],[0.999964,0.00101619,0.00195787,0.00815211]]];
	CONST robtarget pOverPart:=[[-12.15,445.19,84.22],[0.0344175,0.27264,0.961398,0.0139876],[0,-1,1,1],[9E+09,9E+09,9E+09,9E+09,9E+09,9E+09]];
	CONST robtarget pOnPart:=[[-10.40,443.03,33.34],[0.0408588,0.27536,0.960135,0.0254239],[0,-1,0,1],[9E+09,9E+09,9E+09,9E+09,9E+09,9E+09]];
	CONST robtarget pOverConveyor:=[[85.37,-105.04,90.23],[0.0342884,0.272784,0.961361,0.0140776],[-1,-2,1,1],[9E+09,9E+09,9E+09,9E+09,9E+09,9E+09]];
	CONST robtarget pOnConveyor:=[[85.60,-105.21,28.64],[0.0343247,0.272706,0.961384,0.0138928],[-1,-2,1,1],[9E+09,9E+09,9E+09,9E+09,9E+09,9E+09]];
	CONST robtarget pHome:=[[126.23,46.65,186.46],[0.0177685,0.468251,0.793352,-0.388608],[-1,-1,1,1],[9E+09,9E+09,9E+09,9E+09,9E+09,9E+09]];
	CONST robtarget pOverPart2:=[[131.31,460.32,78.64],[0.0343496,0.272936,0.961321,0.0136466],[0,-1,1,1],[9E+09,9E+09,9E+09,9E+09,9E+09,9E+09]];
   CONST robtarget pOnPart2:=[[131.52,460.25,33.28],[0.0344301,0.272923,0.96132,0.0137379],[0,-1,1,1],[9E+09,9E+09,9E+09,9E+09,9E+09,9E+09]];
    CONST robtarget pAtInsp:=[[71.39,122.64,87.02],[0.0343265,0.272697,0.961386,0.0139042],[-1,-1,1,1],[9E+09,9E+09,9E+09,9E+09,9E+09,9E+09]];
   CONST robtarget pNearInsp:=[[61.86,117.36,152.83],[0.0343111,0.272683,0.96139,0.0139106],[-1,-1,1,1],[9E+09,9E+09,9E+09,9E+09,9E+09,9E+09]];
   VAR bool bTimeout:=FALSE;
   VAR num nCount:=0;
   CONST robtarget pOnReject:=[[-46.02,291.57,10.37],[0.034496,0.272705,0.961376,0.0139788],[0,-1,0,1],[9E+09,9E+09,9E+09,9E+09,9E+09,9E+09]];
   CONST robtarget pOverReject:=[[-46.22,291.67,59.56],[0.0344948,0.272701,0.961378,0.0139752],[0,-1,0,1],[9E+09,9E+09,9E+09,9E+09,9E+09,9E+09]];
   CONST robtarget pOverQuench:=[[68.71,143.42,89.77],[0.0343664,0.272942,0.961313,0.0140149],[-1,-1,1,1],[9E+09,9E+09,9E+09,9E+09,9E+09,9E+09]];
   CONST robtarget pOnQuench:=[[68.95,143.28,24.37],[0.0343549,0.27293,0.961317,0.0140139],[-1,-1,1,1],[9E+09,9E+09,9E+09,9E+09,9E+09,9E+09]];
    PROC main()
		MoveJ pHome, v500, fine, tPen\WObj:=wobj1;
        IF DI10_7=1 THEN
		rFeeder1;
    ELSEIF DI10_6=1 THEN
        r_Feeder2;
    ELSE
        RETURN;
    ENDIF
	    rLathe;
        rQuench;
        IF nCount>=3 THEN
            rInspect;
        ELSE
            rConveyor;
        ENDIF
	    RETURN;
	ENDPROC
	PROC rGotoCal()
		MoveAbsJ jposCal\NoEOffs, v1000, z50, tPen\WObj:=wobj1;
	ENDPROC
	PROC rFeeder1()
		MoveJ pOverPart, v500, z30, tPen\WObj:=wobj1;
		MoveL pOnPart, v500, fine, tPen\WObj:=wobj1;
		Set doGrip;
		MoveL pOverPart, v500, z30, tPen\WObj:=wobj1;
		RETURN;
	ENDPROC
	PROC r_Feeder2()
        MoveJ pOverPart2,v500,z30,tPen\WObj:=wobj1;
        MoveL pOnPart2,v500,fine,tPen\WObj:=wobj1;
        Set doGrip;
        MoveL pOverPart2,v500,z30,tPen\WObj:=wobj1;
        RETURN;
    ENDPROC
    PROC rLathe()
		CONST robtarget pOverLathe:=[[286.69,151.67,92.01],[0.0343304,0.27266,0.961396,0.0139257],[-1,-1,1,1],[9E+09,9E+09,9E+09,9E+09,9E+09,9E+09]];
		CONST robtarget pInLathe:=[[286.95,151.53,33.54],[0.0343778,0.272693,0.961386,0.0138903],[-1,-1,1,1],[9E+09,9E+09,9E+09,9E+09,9E+09,9E+09]];
		MoveJ pOverLathe, v500, z10, tPen\WObj:=wobj1;
		MoveL pInLathe, v500, fine, tPen\WObj:=wobj1;
		Reset doGrip;
		MoveL pOverLathe, v500, fine, tPen\WObj:=wobj1;
		PulseDO\PLength:=5, DO10_3;
		WaitDI DI10_5, 1;
		MoveL pInLathe, v500, fine, tPen\WObj:=wobj1;
		Set doGrip;
		MoveJ pOverLathe, v500, z10, tPen\WObj:=wobj1;
        Incr nCount;
        RETURN;
	ENDPROC
    PROC rInspect()
        nCount:=0;
        MoveJ pNearInsp,v500,fine,tPen\WObj:=wobj1;
        MoveJ pAtInsp,v500,fine,tPen\WObj:=wobj1;
        WaitUntil DI10_6=1\MaxTime:=5, \TimeFlag:=bTimeout;
        IF bTimeout=TRUE THEN
            MoveL pOverReject,v500,z30,tPen\WObj:=wobj1;
            MoveL pOnReject,v500,fine,tPen\WObj:=wobj1;
            Reset doGrip;
            MoveL pOverReject,v500,z30,tPen\WObj:=wobj1;
        ELSE
            rConveyor;
        ENDIF
        RETURN;
    ENDPROC
	PROC rConveyor()
		MoveJ pOverConveyor, v500, z60, tPen\WObj:=wobj1;
		MoveL pOnConveyor, v500, fine, tPen\WObj:=wobj1;
		Reset doGrip;
		MoveL pOverConveyor, v500, z60, tPen\WObj:=wobj1;
	ENDPROC
    PROC rQuench()
        MoveJ pOverQuench,v500,z30,tPen\WObj:=wobj1;
        MoveL pOnQuench,v500,fine,tPen\WObj:=wobj1;
        MoveL pOverQuench,v500,z30,tPen\WObj:=wobj1;
        RETURN;
    ENDPROC
ENDMODULE

--- Backups/120-501447/HOME/Conveyor/Lathe/MainModule.mod ---
MODULE MainModule
	TASK PERS tooldata tPen:=[TRUE,[[0.147757,-83.6911,144.451],[0.738156,0.674482,-0.0103991,-0.00950206]],[0.8,[1.7,0,108.7],[1,0,0,0],0.011,0.006,0.009]];
	CONST robtarget p30:=[[469.22,99.75,8.79],[0.0216335,0.64282,0.765703,-0.00355185],[0,0,0,1],[9E+09,9E+09,9E+09,9E+09,9E+09,9E+09]];
	CONST robtarget pstart:=[[512.08,-48.21,10.23],[0.0215519,0.642623,0.765869,-0.00379738],[-1,-1,0,1],[9E+09,9E+09,9E+09,9E+09,9E+09,9E+09]];
	CONST robtarget p10:=[[268.52,32.55,142.20],[0.0387242,0.836099,0.54718,0.00566096],[0,0,0,1],[9E+09,9E+09,9E+09,9E+09,9E+09,9E+09]];
	CONST robtarget p20:=[[268.52,32.55,29.70],[0.0387219,0.8361,0.547177,0.00566567],[0,0,0,1],[9E+09,9E+09,9E+09,9E+09,9E+09,9E+09]];
	CONST robtarget p40:=[[505.98,113.33,4.46],[0.0367854,0.831559,0.554195,0.00482753],[0,0,0,1],[9E+09,9E+09,9E+09,9E+09,9E+09,9E+09]];
	CONST robtarget p50:=[[461.62,115.15,-8.30],[0.0367965,0.831555,0.5542,0.00481934],[0,0,0,1],[9E+09,9E+09,9E+09,9E+09,9E+09,9E+09]];
	CONST robtarget p60:=[[525.97,169.03,3.52],[0.0368121,0.8315,0.554282,0.00472824],[0,0,0,1],[9E+09,9E+09,9E+09,9E+09,9E+09,9E+09]];
	CONST robtarget p70:=[[597.29,115.27,0.65],[0.0368322,0.831492,0.554294,0.00471092],[0,0,0,1],[9E+09,9E+09,9E+09,9E+09,9E+09,9E+09]];
	CONST robtarget p80:=[[569.04,115.26,0.68],[0.036874,0.831516,0.554254,0.00474228],[0,0,0,1],[9E+09,9E+09,9E+09,9E+09,9E+09,9E+09]];
	CONST robtarget p90:=[[579.87,-35.31,-1.57],[0.0368611,0.831471,0.554322,0.00471824],[0,0,0,1],[9E+09,9E+09,9E+09,9E+09,9E+09,9E+09]];
	CONST robtarget p100:=[[547.53,-9.26,-1.58],[0.0368624,0.831474,0.554318,0.00469294],[0,0,0,1],[9E+09,9E+09,9E+09,9E+09,9E+09,9E+09]];
	CONST robtarget p110:=[[532.30,-194.48,243.92],[0.0367212,0.831611,0.55412,0.00498134],[-1,0,0,1],[9E+09,9E+09,9E+09,9E+09,9E+09,9E+09]];
	TASK PERS wobjdata wFixture1:=[FALSE,TRUE,"",[[0,0,0],[1,0,0,0]],[[357.689,-176.134,-17.7192],[0.999991,-0.00111829,0.000705852,-0.00392021]]];
	TASK PERS wobjdata wobj1:=[FALSE,TRUE,"",[[0,0,0],[1,0,0,0]],[[372.049,-59.0817,-2.31291],[0.999964,0.00101619,0.00195787,0.00815211]]];
	CONST robtarget pOverPart:=[[-12.15,445.19,84.22],[0.0344175,0.27264,0.961398,0.0139876],[0,-1,1,1],[9E+09,9E+09,9E+09,9E+09,9E+09,9E+09]];
	CONST robtarget pOnPart:=[[-10.40,443.03,33.34],[0.0408588,0.27536,0.960135,0.0254239],[0,-1,0,1],[9E+09,9E+09,9E+09,9E+09,9E+09,9E+09]];
	PROC main()
		MoveJ p10, v1000, z50, tPen\WObj:=wobj1;
		MoveL p20, v1000, fine, tPen\WObj:=wobj1;
		Set doGrip;
		MoveL p10, v1000, fine, tPen\WObj:=wobj1;
		MoveL [[523.80,-56.63,-8.74],[0.0367413,0.831596,0.554142,0.00493633],[0,0,0,1],[9E+09,9E+09,9E+09,9E+09,9E+09,9E+09]], v1000, fine, tPen\WObj:=wobj1;
		MoveL [[449.04,-57.95,-7.57],[0.0367587,0.831587,0.554155,0.00488328],[0,0,1,1],[9E+09,9E+09,9E+09,9E+09,9E+09,9E+09]], v1000, fine, tPen\WObj:=wobj1;
		MoveL [[497.17,94.80,-7.58],[0.0367718,0.831577,0.554169,0.00486949],[0,0,0,1],[9E+09,9E+09,9E+09,9E+09,9E+09,9E+09]], v1000, fine, tPen\WObj:=wobj1;
		MoveL [[524.39,-59.04,-6.34],[0.037286,0.83168,0.553975,0.00527583],[0,0,0,1],[9E+09,9E+09,9E+09,9E+09,9E+09,9E+09]], v1000, fine, tPen\WObj:=wobj1;
		MoveL p10, v1000, fine, tPen;
		MoveL p20, v1000, fine, tPen;
		Reset doGrip;
	ENDPROC
	PROC rGotoCal()
		MoveAbsJ jposCal\NoEOffs, v1000, z50, tPen\WObj:=wobj1;
	ENDPROC
	PROC rFeeder1()
		MoveJ pOverPart, v500, z30, tPen\WObj:=wobj1;
		MoveL pOnPart, v500, fine, tPen\WObj:=wobj1;
		Set doGrip;
		MoveL pOverPart, v500, z30, tPen\WObj:=wobj1;
		RETURN;
	ENDPROC
	PROC rLathe()
		CONST robtarget pOverLathe:=[[286.69,151.67,92.01],[0.0343304,0.27266,0.961396,0.0139257],[-1,-1,1,1],[9E+09,9E+09,9E+09,9E+09,9E+09,9E+09]];
		CONST robtarget pInLathe:=[[286.95,151.53,33.54],[0.0343778,0.272693,0.961386,0.0138903],[-1,-1,1,1],[9E+09,9E+09,9E+09,9E+09,9E+09,9E+09]];
		MoveJ pOverLathe, v500, z10, tPen\WObj:=wobj1;
		MoveL pInLathe, v500, fine, tPen\WObj:=wobj1;
		Reset doGrip;
		MoveL pOverLathe, v500, fine, tPen\WObj:=wobj1;
		PulseDO\PLength:=5, DO10_3;
		WaitDI DI10_5, 1;
		MoveL pInLathe, v500, fine, tPen\WObj:=wobj1;
		Set doGrip;
		MoveJ pOverLathe, v500, z10, tPen\WObj:=wobj1;
	ENDPROC
ENDMODULE

--- Backups/120-501447/HOME/Happy/MainModule.mod ---
MODULE MainModule
	TASK PERS tooldata toolpen:=[TRUE,[[1.46446,-97.4412,143.449],[0.707234,0.706949,0.00461643,0.00461459]],[0.9,[1.9,0,87.7],[1,0,0,0],0.018,0.014,0.009]];
	CONST jointtarget jpos10:=[[0,0,0,0,0,0],[9E+09,9E+09,9E+09,9E+09,9E+09,9E+09]];
	TASK PERS tooldata toolgrip:=[TRUE,[[0.33438,5.55227,149.366],[0.707192,0.706991,0.00466561,0.00466421]],[0.9,[1.9,0,87.7],[1,0,0,0],0,0,0]];
	TASK PERS tooldata toolsuck:=[TRUE,[[0.737948,-50.1456,37.5188],[0.707214,0.706968,0.00471148,0.0047099]],[0.9,[1.9,0,87.7],[1,0,0,0],0,0,0]];
	TASK PERS wobjdata wobjgraph:=[FALSE,TRUE,"",[[0,0,0],[1,0,0,0]],[[273.288,-283.326,55.6201],[0.999877,-2.17942E-06,-4.90728E-06,-0.0157116]]];
	CONST robtarget home:=[[623.25,3.42,336.16],[0.0299097,0.676932,0.735397,0.00769099],[-1,-1,1,1],[9E+09,9E+09,9E+09,9E+09,9E+09,9E+09]];
	VAR num command:=0;
    VAR num firstpass:=0;
    VAR errnum errvar;
    VAR intnum drop:=0;
	CONST robtarget yes_up:=[[636.61,12.86,390.65],[0.110766,0.65786,0.738846,0.0951692],[-1,-1,1,1],[9E+09,9E+09,9E+09,9E+09,9E+09,9E+09]];
	CONST robtarget yes_down:=[[587.20,-9.01,273.39],[0.0750995,-0.686949,-0.71509,0.105386],[-1,-1,1,1],[9E+09,9E+09,9E+09,9E+09,9E+09,9E+09]];
    CONST robtarget no_left:=[[613.43,110.32,335.98],[0.0290328,0.611086,0.790966,0.0101249],[0,-1,1,1],[9E+09,9E+09,9E+09,9E+09,9E+09,9E+09]];
    CONST robtarget no_right:=[[609.66,-129.55,335.98],[0.0304386,0.751885,0.658576,0.00434813],[-1,-1,1,1],[9E+09,9E+09,9E+09,9E+09,9E+09,9E+09]];
	CONST robtarget look_left_home:=[[240.90,431.80,554.59],[0.0290953,-0.281789,-0.937121,0.203843],[0,-1,1,0],[9E+09,9E+09,9E+09,9E+09,9E+09,9E+09]];
	CONST robtarget look_left_home10:=[[202.32,462.83,563.63],[0.270093,-0.324969,-0.897791,0.12416],[0,-1,1,0],[9E+09,9E+09,9E+09,9E+09,9E+09,9E+09]];
	CONST robtarget look_left_home20:=[[270.63,415.58,562.23],[0.138289,0.240897,0.92733,-0.250804],[0,-1,0,0],[9E+09,9E+09,9E+09,9E+09,9E+09,9E+09]];
	CONST robtarget look_left_home30:=[[270.64,415.58,562.21],[0.1734,0.215279,0.956874,-0.0893234],[0,0,0,0],[9E+09,9E+09,9E+09,9E+09,9E+09,9E+09]];
	CONST robtarget look_left_home40:=[[270.64,415.58,562.21],[0.139813,0.245163,0.920572,-0.269988],[0,-1,0,0],[9E+09,9E+09,9E+09,9E+09,9E+09,9E+09]];
	CONST robtarget POKE:=[[355.93,589.27,233.27],[0.139842,0.245165,0.92056,-0.270011],[0,-1,1,0],[9E+09,9E+09,9E+09,9E+09,9E+09,9E+09]];
	CONST robtarget clap_home:=[[361.01,-7.97,835.78],[0.227814,0.709062,0.667087,0.0180613],[0,-1,0,2],[9E+09,9E+09,9E+09,9E+09,9E+09,9E+09]];
	CONST robtarget clap_1:=[[432.72,24.08,749.46],[0.0784551,0.705231,0.704216,-0.0239353],[0,-1,0,2],[9E+09,9E+09,9E+09,9E+09,9E+09,9E+09]];
	CONST robtarget home10:=[[440.55,186.95,302.74],[0.054125,-0.114661,-0.990357,0.0558274],[-1,-1,1,1],[9E+09,9E+09,9E+09,9E+09,9E+09,9E+09]];
	CONST robtarget stare_left:=[[476.96,208.62,340.44],[0.0133216,0.164619,0.985642,0.0351197],[-1,-1,1,1],[9E+09,9E+09,9E+09,9E+09,9E+09,9E+09]];
	CONST robtarget home20:=[[623.67,20.06,341.98],[0.0571571,-0.683156,-0.721013,-0.100851],[-1,-1,1,1],[9E+09,9E+09,9E+09,9E+09,9E+09,9E+09]];
	CONST robtarget rockout:=[[623.67,20.07,341.98],[0.0571572,-0.683155,-0.721014,-0.100851],[-1,-1,1,1],[9E+09,9E+09,9E+09,9E+09,9E+09,9E+09]];
	CONST robtarget rockout10:=[[626.14,-70.04,367.53],[0.296474,0.647388,0.659861,-0.239947],[-1,-1,0,1],[9E+09,9E+09,9E+09,9E+09,9E+09,9E+09]];
	CONST robtarget rockout20:=[[270.61,12.44,724.40],[0.110762,-0.706757,-0.697822,0.0356268],[0,-1,1,2],[9E+09,9E+09,9E+09,9E+09,9E+09,9E+09]];
	CONST robtarget rockout30:=[[270.61,12.44,724.40],[0.115213,-0.577315,-0.80819,0.0162022],[-1,0,0,2],[9E+09,9E+09,9E+09,9E+09,9E+09,9E+09]];
	CONST robtarget rockout40:=[[562.15,-152.86,603.28],[0.0379782,-0.747438,-0.663244,0.000773863],[-1,0,0,0],[9E+09,9E+09,9E+09,9E+09,9E+09,9E+09]];
	CONST robtarget rockout50:=[[562.15,-152.87,603.27],[0.0930603,-0.73457,-0.655846,-0.147013],[-1,0,0,0],[9E+09,9E+09,9E+09,9E+09,9E+09,9E+09]];
	CONST robtarget rockout60:=[[562.15,-152.87,603.27],[0.21023,0.722718,0.628168,-0.197196],[-1,0,0,0],[9E+09,9E+09,9E+09,9E+09,9E+09,9E+09]];
	CONST robtarget rockout70:=[[562.16,-152.87,603.27],[0.148229,0.737836,0.607969,-0.252978],[-1,-1,0,0],[9E+09,9E+09,9E+09,9E+09,9E+09,9E+09]];
	CONST robtarget rockout80:=[[520.54,-149.29,575.14],[0.14822,0.737835,0.607971,-0.252983],[-1,-1,0,0],[9E+09,9E+09,9E+09,9E+09,9E+09,9E+09]];
	CONST robtarget rockout90:=[[367.81,-148.61,575.15],[0.148223,0.737831,0.607972,-0.252991],[-1,0,0,0],[9E+09,9E+09,9E+09,9E+09,9E+09,9E+09]];
	CONST robtarget rockout100:=[[637.88,-134.02,250.68],[0.0430323,-0.78077,-0.620734,0.056874],[-1,0,0,1],[9E+09,9E+09,9E+09,9E+09,9E+09,9E+09]];
	CONST robtarget rockout110:=[[637.88,-134.02,250.68],[0.177143,-0.771197,-0.597683,-0.129039],[-1,-1,1,1],[9E+09,9E+09,9E+09,9E+09,9E+09,9E+09]];
	CONST robtarget rockout120:=[[637.88,-134.02,250.68],[0.0094828,-0.791224,-0.556696,-0.252911],[-1,0,1,1],[9E+09,9E+09,9E+09,9E+09,9E+09,9E+09]];
	CONST robtarget rockout130:=[[637.88,-134.02,250.68],[0.0496911,0.770261,0.577791,-0.265304],[-1,0,0,1],[9E+09,9E+09,9E+09,9E+09,9E+09,9E+09]];
	CONST robtarget rockout140:=[[637.88,-134.02,250.68],[0.0139427,0.68655,0.675124,-0.26956],[-1,-1,0,1],[9E+09,9E+09,9E+09,9E+09,9E+09,9E+09]];
	CONST robtarget rockout150:=[[637.88,-134.02,250.67],[0.172983,0.681723,0.698718,-0.130852],[-1,-1,0,1],[9E+09,9E+09,9E+09,9E+09,9E+09,9E+09]];
	CONST robtarget rockout160:=[[637.87,-134.02,250.68],[0.0181335,0.70293,0.652008,-0.283629],[-1,0,0,1],[9E+09,9E+09,9E+09,9E+09,9E+09,9E+09]];
	CONST robtarget rockout170:=[[223.26,-26.70,704.77],[0.118778,-0.734568,-0.658528,0.112436],[-1,0,0,0],[9E+09,9E+09,9E+09,9E+09,9E+09,9E+09]];
	CONST robtarget rockout180:=[[128.96,-184.19,704.76],[0.154334,-0.939388,-0.301326,0.0541592],[-1,0,0,0],[9E+09,9E+09,9E+09,9E+09,9E+09,9E+09]];
	CONST robtarget rockout190:=[[97.93,202.40,704.76],[0.0314087,-0.215609,-0.962684,0.160514],[0,0,0,0],[9E+09,9E+09,9E+09,9E+09,9E+09,9E+09]];
	CONST robtarget rockout200:=[[228.08,-23.75,474.40],[0.11875,-0.734577,-0.658522,0.112439],[-1,-1,1,0],[9E+09,9E+09,9E+09,9E+09,9E+09,9E+09]];
	CONST robtarget rockout210:=[[228.08,-76.46,474.40],[0.118752,-0.734578,-0.658521,0.112437],[-1,0,0,0],[9E+09,9E+09,9E+09,9E+09,9E+09,9E+09]];
	CONST robtarget rockout220:=[[228.08,21.44,474.40],[0.118747,-0.734574,-0.658526,0.112439],[0,-1,1,0],[9E+09,9E+09,9E+09,9E+09,9E+09,9E+09]];
	CONST robtarget rockout230:=[[-30.60,-167.76,770.60],[0.00191724,-0.997314,0.0689616,0.0245916],[-2,-1,0,6],[9E+09,9E+09,9E+09,9E+09,9E+09,9E+09]];
	CONST robtarget rockout240:=[[-8.27,-499.51,476.38],[0.108981,-0.994002,0.00891335,0.00165642],[-2,-1,1,0],[9E+09,9E+09,9E+09,9E+09,9E+09,9E+09]];
	CONST robtarget rockout250:=[[4.31,-338.46,434.02],[0.101452,-0.994816,-0.00617029,0.00324005],[-1,-1,1,0],[9E+09,9E+09,9E+09,9E+09,9E+09,9E+09]];
	CONST robtarget rockout260:=[[-30.60,-167.76,770.60],[0.00191718,-0.997313,0.0689699,0.0245909],[-2,-1,0,6],[9E+09,9E+09,9E+09,9E+09,9E+09,9E+09]];
	CONST robtarget rockout270:=[[-39.44,-323.02,739.67],[0.0149149,-0.997603,0.0505067,0.0448726],[-2,-1,0,0],[9E+09,9E+09,9E+09,9E+09,9E+09,9E+09]];
	CONST robtarget rockout280:=[[20.47,170.78,770.08],[0.0246627,0.0388613,0.998936,-0.00271462],[0,-1,0,6],[9E+09,9E+09,9E+09,9E+09,9E+09,9E+09]];
	CONST robtarget home30:=[[20.47,170.78,770.08],[0.0246627,0.0388613,0.998936,-0.00271462],[0,-1,0,6],[9E+09,9E+09,9E+09,9E+09,9E+09,9E+09]];
	CONST robtarget rockout290:=[[17.26,266.75,764.82],[0.0238403,0.0269462,0.999352,-0.00124431],[0,-1,0,0],[9E+09,9E+09,9E+09,9E+09,9E+09,9E+09]];
	CONST string max_time:="";
	CONST robtarget home40:=[[698.66,235.47,87.29],[0.267708,-0.617083,-0.68548,-0.27867],[0,0,1,1],[9E+09,9E+09,9E+09,9E+09,9E+09,9E+09]];
	CONST robtarget doink_pickup:=[[389.45,502.54,-21.58],[0.331101,-0.728834,-0.593014,-0.0866466],[0,0,0,1],[9E+09,9E+09,9E+09,9E+09,9E+09,9E+09]];
	CONST robtarget doink_pickup10:=[[-101.82,420.19,21.86],[0.379294,0.00755716,-0.924909,0.0249635],[0,-1,1,1],[9E+09,9E+09,9E+09,9E+09,9E+09,9E+09]];
	CONST robtarget doink_pickup1:=[[-92.11,418.52,45.28],[0.379241,0.00760408,-0.92493,0.0249756],[0,-1,1,1],[9E+09,9E+09,9E+09,9E+09,9E+09,9E+09]];
	CONST robtarget doink_pickup11:=[[-153.15,-39.95,547.97],[0.254139,0.96068,0.0368876,0.105581],[-1,0,0,1],[9E+09,9E+09,9E+09,9E+09,9E+09,9E+09]];
	CONST robtarget doink_pickup21:=[[407.26,-190.36,716.04],[0.193083,0.866404,0.414882,0.199838],[-1,0,0,1],[9E+09,9E+09,9E+09,9E+09,9E+09,9E+09]];
	CONST robtarget doink_pickup31:=[[-47.62,592.06,370.04],[0.0580329,0.32425,0.943871,0.0245335],[0,0,0,1],[9E+09,9E+09,9E+09,9E+09,9E+09,9E+09]];
	CONST robtarget doink_pickup41:=[[16.75,722.64,270.38],[0.0580336,0.324246,0.943872,0.0245342],[0,0,0,1],[9E+09,9E+09,9E+09,9E+09,9E+09,9E+09]];
	CONST robtarget scratch:=[[61.65,-39.90,132.58],[0.507371,-0.0115254,-0.795923,0.330072],[-1,-2,1,1],[9E+09,9E+09,9E+09,9E+09,9E+09,9E+09]];
	CONST robtarget scratch10:=[[50.52,-42.75,138.78],[0.529894,0.0183839,-0.788381,0.311976],[-1,-2,1,1],[9E+09,9E+09,9E+09,9E+09,9E+09,9E+09]];
	CONST robtarget scratch20:=[[61.91,-57.03,114.11],[0.506617,-0.0326626,-0.784616,0.355878],[-1,-2,1,1],[9E+09,9E+09,9E+09,9E+09,9E+09,9E+09]];
	CONST robtarget scratch30:=[[210.45,194.50,146.34],[0.388587,-0.0926191,-0.913366,0.0786347],[-1,-1,1,1],[9E+09,9E+09,9E+09,9E+09,9E+09,9E+09]];
	CONST robtarget stare_left_cock:=[[471.21,193.05,328.12],[0.0169203,0.148751,0.988727,-0.00243101],[-1,-1,1,1],[9E+09,9E+09,9E+09,9E+09,9E+09,9E+09]];
	CONST robtarget stare_left10:=[[434.18,222.49,350.76],[0.220401,-0.151719,-0.960761,-0.0730921],[-1,-1,1,1],[9E+09,9E+09,9E+09,9E+09,9E+09,9E+09]];
	CONST robtarget stare_left20:=[[507.37,197.73,346.36],[0.179179,0.168109,0.969323,0.00687501],[-1,-1,1,1],[9E+09,9E+09,9E+09,9E+09,9E+09,9E+09]];
	CONST robtarget stare_left30:=[[232.46,2.83,31.19],[0.17951,-0.905593,0.337486,-0.183792],[0,1,1,1],[9E+09,9E+09,9E+09,9E+09,9E+09,9E+09]];
	CONST robtarget stare_left40:=[[215.15,-13.26,52.77],[0.116753,-0.918091,0.342409,-0.161967],[0,1,1,1],[9E+09,9E+09,9E+09,9E+09,9E+09,9E+09]];
	CONST robtarget lick1:=[[215.15,-13.26,52.77],[0.116753,-0.918091,0.342409,-0.161967],[0,1,1,1],[9E+09,9E+09,9E+09,9E+09,9E+09,9E+09]];
	CONST robtarget lick11:=[[237.45,7.63,25.86],[0.196495,-0.901457,0.335879,-0.189602],[0,1,1,1],[9E+09,9E+09,9E+09,9E+09,9E+09,9E+09]];
	CONST robtarget stare_left50:=[[431.13,460.69,268.14],[0.08496,-0.374212,-0.915851,0.11817],[0,0,1,1],[9E+09,9E+09,9E+09,9E+09,9E+09,9E+09]];
	CONST robtarget look_at_feeder:=[[431.13,460.69,268.14],[0.0849594,-0.374212,-0.91585,0.118173],[0,0,1,1],[9E+09,9E+09,9E+09,9E+09,9E+09,9E+09]];
	CONST robtarget look_at_feeder10:=[[407.13,436.45,235.56],[0.121129,-0.369158,-0.897353,0.2093],[0,0,1,1],[9E+09,9E+09,9E+09,9E+09,9E+09,9E+09]];
	CONST robtarget look_at_feeder20:=[[627.45,84.59,395.10],[0.00347987,0.669314,0.742868,-0.0123751],[0,0,0,1],[9E+09,9E+09,9E+09,9E+09,9E+09,9E+09]];
	CONST robtarget look_at_feeder30:=[[627.45,-305.71,395.10],[0.00348066,0.669316,0.742867,-0.0123764],[-1,-1,1,1],[9E+09,9E+09,9E+09,9E+09,9E+09,9E+09]];
	CONST robtarget look_at_feeder40:=[[630.79,326.98,395.10],[0.00348235,0.669315,0.742867,-0.0123759],[0,0,0,1],[9E+09,9E+09,9E+09,9E+09,9E+09,9E+09]];
	CONST robtarget look_at_feeder50:=[[562.52,-56.08,395.08],[0.00347547,0.669318,0.742864,-0.0123909],[-1,-1,1,1],[9E+09,9E+09,9E+09,9E+09,9E+09,9E+09]];
	CONST robtarget stare_left60:=[[476.96,208.63,340.44],[0.0327909,0.161855,0.974473,0.152081],[-1,-1,1,1],[9E+09,9E+09,9E+09,9E+09,9E+09,9E+09]];
	CONST robtarget look_up_dn1:=[[476.95,208.63,340.43],[0.0327917,0.161852,0.974474,0.152078],[-1,-1,1,1],[9E+09,9E+09,9E+09,9E+09,9E+09,9E+09]];
	CONST robtarget look_up_dn11:=[[476.95,208.63,340.43],[0.034403,-0.161391,-0.952917,0.254399],[0,-2,2,1],[9E+09,9E+09,9E+09,9E+09,9E+09,9E+09]];
	CONST robtarget look_up_dn21:=[[476.95,208.62,340.44],[0.188679,0.0964486,0.933725,-0.288539],[0,-2,1,1],[9E+09,9E+09,9E+09,9E+09,9E+09,9E+09]];
	CONST robtarget look_up_dn31:=[[476.96,208.62,340.43],[0.118405,0.101949,0.985432,-0.0671546],[0,-1,1,1],[9E+09,9E+09,9E+09,9E+09,9E+09,9E+09]];
	CONST robtarget look_up_dn41:=[[476.96,208.63,340.43],[0.991171,-0.0583428,-0.0575373,-0.104237],[-1,-1,3,1],[9E+09,9E+09,9E+09,9E+09,9E+09,9E+09]];
	CONST robtarget look_up_dn51:=[[476.96,208.62,340.44],[0.00911973,0.106958,0.992798,-0.0531872],[0,-1,1,1],[9E+09,9E+09,9E+09,9E+09,9E+09,9E+09]];
	CONST robtarget doink_pickup51:=[[42.19,482.69,261.79],[0.278798,-0.687523,-0.630227,-0.228906],[0,0,1,1],[9E+09,9E+09,9E+09,9E+09,9E+09,9E+09]];
	CONST robtarget above_play:=[[566.77,-37.05,-2.71],[0.0428487,0.625954,0.74184,-0.236684],[-1,-1,0,1],[9E+09,9E+09,9E+09,9E+09,9E+09,9E+09]];
	CONST robtarget press_play:=[[566.78,-37.04,-17.09],[0.0428818,0.625936,0.741858,-0.236668],[-1,-1,0,1],[9E+09,9E+09,9E+09,9E+09,9E+09,9E+09]];
	CONST robtarget above_play10:=[[566.77,-37.05,-2.71],[0.0428487,0.625954,0.74184,-0.236684],[-1,-1,0,1],[9E+09,9E+09,9E+09,9E+09,9E+09,9E+09]];
	CONST robtarget doink_pickup71:=[[476.96,208.62,340.43],[0.0133153,0.164616,0.985642,0.0351121],[-1,-1,1,1],[9E+09,9E+09,9E+09,9E+09,9E+09,9E+09]];
	CONST robtarget doink_pickup61:=[[103.04,-437.58,716.05],[0.260895,0.960605,-0.00437255,0.0956642],[-1,0,0,1],[9E+09,9E+09,9E+09,9E+09,9E+09,9E+09]];
	CONST robtarget doink_pickup91:=[[56.72,351.84,641.66],[0.109346,-0.596771,-0.620099,-0.497378],[0,0,0,1],[9E+09,9E+09,9E+09,9E+09,9E+09,9E+09]];
	CONST robtarget doink_pickup81:=[[4.69,83.51,591.11],[0.150037,0.86147,0.329378,0.356187],[-1,0,0,1],[9E+09,9E+09,9E+09,9E+09,9E+09,9E+09]];
	CONST robtarget doink_pickup20:=[[143.07,289.22,517.39],[0.0663871,0.69878,0.708174,0.0760855],[0,0,0,1],[9E+09,9E+09,9E+09,9E+09,9E+09,9E+09]];
	CONST robtarget cupdrop1:=[[143.07,289.22,517.39],[0.0663889,0.69878,0.708174,0.0760848],[0,0,0,1],[9E+09,9E+09,9E+09,9E+09,9E+09,9E+09]];
	CONST robtarget cupdrop21:=[[-10.85,81.56,517.38],[0.0868058,0.885084,0.454357,0.0514952],[-1,0,0,1],[9E+09,9E+09,9E+09,9E+09,9E+09,9E+09]];
	CONST robtarget cupdrop11:=[[-10.85,81.56,517.37],[0.0868013,0.885086,0.454356,0.0514711],[-1,0,0,1],[9E+09,9E+09,9E+09,9E+09,9E+09,9E+09]];
	CONST jointtarget jpos20:=[[-60,0.141048,5.45631,5.41479,-17.2219,84.4552],[9E+09,9E+09,9E+09,9E+09,9E+09,9E+09]];
	CONST jointtarget jpos30:=[[60,0.141048,5.45631,5.41479,-17.2219,84.4552],[9E+09,9E+09,9E+09,9E+09,9E+09,9E+09]];

	TASK PERS wobjdata setup:=[FALSE,TRUE,"",[[385.823,-290.147,8.50775],[1,5.95867E-07,1.00424E-05,-5.95105E-06]],[[0,0,0],[1,0,0,0]]];
	CONST robtarget setuphome:=[[45.60,86.26,94.38],[7.9049E-05,0.954176,0.299245,0.00015283],[-1,0,0,1],[9E+09,9E+09,9E+09,9E+09,9E+09,9E+09]];
    CONST robtarget setup_aboveframe:=[[31.22,63.25,34.24],[0.0507358,-0.947263,-0.312647,-0.048677],[-1,0,1,1],[9E+09,9E+09,9E+09,9E+09,9E+09,9E+09]];
    CONST robtarget setup_aboveseat_load1:=[[84.51,52.57,38.91],[0.0507381,-0.947263,-0.312646,-0.0486824],[-1,0,0,1],[9E+09,9E+09,9E+09,9E+09,9E+09,9E+09]];
    CONST robtarget setup_atseat_load1:=[[93.09,50.89,9.10],[0.0865402,-0.940794,-0.326714,-0.0259962],[-1,0,0,1],[9E+09,9E+09,9E+09,9E+09,9E+09,9E+09]];
    CONST robtarget setup_abovebody_load2:=[[155.09,88.56,74.41],[0.112268,-0.878329,-0.459848,-0.0668867],[-1,0,1,1],[9E+09,9E+09,9E+09,9E+09,9E+09,9E+09]];
    CONST robtarget setup_atbody_load2:=[[159.72,88.56,20.11],[0.0504336,-0.88311,-0.466431,-0.00386496],[-1,0,0,1],[9E+09,9E+09,9E+09,9E+09,9E+09,9E+09]];
    CONST robtarget setup_place_seat:=[[45.60,86.26,94.38],[7.9049E-05,0.954176,0.299245,0.00015283],[-1,0,0,1],[9E+09,9E+09,9E+09,9E+09,9E+09,9E+09]];
     CONST robtarget setup_place_body:=[[45.60,86.26,94.38],[7.9049E-05,0.954176,0.299245,0.00015283],[-1,0,0,1],[9E+09,9E+09,9E+09,9E+09,9E+09,9E+09]];
     CONST robtarget setup_aboveseat_badload3:=[[45.60,86.26,94.38],[7.9049E-05,0.954176,0.299245,0.00015283],[-1,0,0,1],[9E+09,9E+09,9E+09,9E+09,9E+09,9E+09]];
    CONST robtarget setup_atseat_badload3:=[[45.60,86.26,94.38],[7.9049E-05,0.954176,0.299245,0.00015283],[-1,0,0,1],[9E+09,9E+09,9E+09,9E+09,9E+09,9E+09]];
    CONST robtarget setup_abovebody_badload4:=[[45.60,86.26,94.38],[7.9049E-05,0.954176,0.299245,0.00015283],[-1,0,0,1],[9E+09,9E+09,9E+09,9E+09,9E+09,9E+09]];
  CONST robtarget setup_place_seat_on_frame:=[[31.21,63.25,11.34],[0.0507362,-0.947264,-0.312645,-0.0486779],[-1,0,1,1],[9E+09,9E+09,9E+09,9E+09,9E+09,9E+09]];
   CONST robtarget setup_place_body_on_frame:=[[35.89,96.30,21.42],[0.00408463,-0.893244,-0.449449,-0.00971498],[-1,0,0,1],[9E+09,9E+09,9E+09,9E+09,9E+09,9E+09]];
	CONST robtarget setup_body_above_frame:=[[35.89,96.29,92.19],[0.00408465,-0.893246,-0.449445,-0.00971406],[-1,0,0,1],[9E+09,9E+09,9E+09,9E+09,9E+09,9E+09]];
	  VAR num clockdata:=0;
	  CONST robtarget setup_above_pen:=[[181.23,-164.85,147.67],[0.00695138,-0.953914,-0.299993,-0.00178233],[-1,0,0,1],[9E+09,9E+09,9E+09,9E+09,9E+09,9E+09]];
       CONST robtarget setup_at_pen:=[[181.23,-164.85,-8.14],[0.00695467,-0.953914,-0.299994,-0.001786],[-1,0,0,1],[9E+09,9E+09,9E+09,9E+09,9E+09,9E+09]];
       CONST robtarget setup_pen_above_frame:=[[34.25,102.80,53.44],[0.0201754,-0.953182,-0.301712,0.00256073],[-1,0,0,1],[9E+09,9E+09,9E+09,9E+09,9E+09,9E+09]];
       CONST robtarget setup_pen_glue1_frame:=[[34.25,102.80,53.44],[0.17595,-0.925377,-0.328187,-0.0707928],[-1,0,1,1],[9E+09,9E+09,9E+09,9E+09,9E+09,9E+09]];
       CONST robtarget setup_pen_glue2_frame:=[[34.25,102.80,53.44],[0.0943029,-0.911616,-0.340973,-0.209287],[-1,0,1,1],[9E+09,9E+09,9E+09,9E+09,9E+09,9E+09]];
       CONST robtarget setup_pen_glue3_frame:=[[34.25,102.80,53.44],[0.010372,0.892905,0.388022,-0.228147],[-1,0,0,1],[9E+09,9E+09,9E+09,9E+09,9E+09,9E+09]];
       CONST robtarget setup_pen_glue4_frame:=[[34.25,102.80,53.44],[0.0956252,0.889619,0.408975,-0.179368],[-1,0,0,1],[9E+09,9E+09,9E+09,9E+09,9E+09,9E+09]];
       CONST robtarget setup_pen_glue5_frame:=[[15.65,94.76,28.01],[0.0539684,-0.917631,-0.393745,0.00212898],[-1,0,1,1],[9E+09,9E+09,9E+09,9E+09,9E+09,9E+09]];
    CONST robtarget setup_pen_glue6_frame:=[[15.65,121.33,28.02],[0.0539588,-0.917631,-0.393748,0.00211925],[-1,0,1,1],[9E+09,9E+09,9E+09,9E+09,9E+09,9E+09]];
   CONST robtarget setup_pen_glue7_frame:=[[43.03,118.23,28.01],[0.0539597,-0.917632,-0.393746,0.00212379],[-1,0,1,1],[9E+09,9E+09,9E+09,9E+09,9E+09,9E+09]];
   CONST robtarget setup_pen_glue8_frame:=[[43.03,94.73,28.02],[0.0539608,-0.917633,-0.393743,0.00212307],[-1,0,1,1],[9E+09,9E+09,9E+09,9E+09,9E+09,9E+09]];
   PROC main()
          !! Intrrupt for vac to drop ball	the if then connects var drop with vacdrop now only once during first run
            IF firstpass=0 THEN
            	CONNECT drop WITH VacDropNow;
                ISignalDI DI10_9, 1, drop;
                 ISleep drop;
           ENDIF
            Incr firstpass;
         ISleep drop;
        MoveJ stare_left, v300, z150, toolpen;
        Reset DO10_14;
        Reset doGrip;
        Reset doVacume;
        TPErase;
		TPReadFK command, "WHAT DO YOU WANT ME TO DO MENU 1", "YES", "NO", "LOOK LEFT", "CLAP", "MORE";
        TEST command
        CASE 1:
        yes;
        CASE 2:
        no;
        CASE 3:
        look_left;
        CASE 4:
       clap;
        CASE 5:
        GOTO NEXT;
        ENDTEST
        NEXT:
        Reset DO10_14;
        TPReadFK command, "WHAT DO YOU WANT ME TO DO MENU 2", "ROCK OUT", "CLAP", "Snake Strike", "THROW BALL", "MORE";
        TEST command
        CASE 1:
        rock_out;
        CASE 2:
        clap;
        CASE 3:
        photo_activate;
        CASE 4:
        PONG_DOINK;
        CASE 5:
       GOTO NEXT1;
        ENDTEST
        NEXT1:
        Reset DO10_14;
        TPReadFK command, "WHAT DO YOU WANT ME TO DO MENU 3", "PLAY MUSIC", "LOOK ABOUT", "CUP DROP", "SCRATCH", "MORE";
        TEST command
        CASE 1:
        PLAY_MUSIC;
        CASE 2:
       LOOK_ABOUT;
        CASE 3:
        CupDrop;
        CASE 4:
        SCRATCH1;
        CASE 5:
        GOTO NEXT2;
        ENDTEST
        NEXT2:
        Reset DO10_14;
        TPReadFK command, "WHAT DO YOU WANT ME TO DO MENU 4", "BALL MADNESS", "LICK", "COCK HEAD", "DEMO", "MORE";
        TEST command
        CASE 1:
        BALL_MADNESS;
        CASE 2:
        LICK;
        CASE 3:
        COCK_HEAD;
        CASE 4:
       DEMO;
        CASE 5:
       GOTO NEXT3;
        ENDTEST
        NEXT3:
           Reset DO10_14;
        TPReadFK command, "WHAT DO YOU WANT ME TO DO MENU 4", "BUILD CAR", "LICK", "COCK HEAD", "DEMO", "MENU 1";
        TEST command
        CASE 1:
        setup_RED;
        CASE 2:
        LICK;
        CASE 3:
        COCK_HEAD;
        CASE 4:
       DEMO;
        CASE 5:
       main;
        ENDTEST

	ENDPROC
	PROC yes()
		MoveJ home, v1000, z50, toolpen;
        Set DO10_14;
		MoveJ yes_down, v1000, z50, toolpen;
		MoveJ yes_up, v1000, z50, toolpen;
        MoveJ yes_down, v1000, z50, toolpen;
		MoveJ yes_up, v1000, z50, toolpen;
        MoveJ yes_down, v1000, z50, toolpen;
		MoveJ yes_up, v1000, z50, toolpen;
        MoveJ home, v1000, z50, toolpen;
	    main;
	ENDPROC
	PROC no()
		MoveJ home, v1000, z50, toolpen;
        Set DO10_14;
		MoveJ no_left, v1000, z50, toolpen;
		MoveJ no_right, v1000, z50, toolpen;
        MoveJ no_left, v1000, z50, toolpen;
		MoveJ no_right, v1000, z50, toolpen;
        MoveJ no_left, v1000, z50, toolpen;
		MoveJ no_right, v1000, z50, toolpen;
        MoveJ home, v1000, z50, toolpen;
        main;
	ENDPROC
	PROC look_left()
		MoveJ look_left_home, v500, z50, toolpen;
		MoveJ look_left_home10, v100, fine, toolpen;
        Set doGrip;
        WaitTime .5;
        Reset doGrip;
        WaitTime .5;
		MoveJ look_left_home20, v100, fine, toolpen;
         Set doGrip;
        WaitTime .5;
        Reset doGrip;
        WaitTime .5;
        Set DO10_14;
        WaitTime 1;
        Reset DO10_14;
        WaitTime 1;
        MoveJ look_left_home30, v100, fine, toolpen;
        MoveJ look_left_home40, v100, fine, toolpen;
        TPReadFK command, "Poke When Photo Eye Made?", "YES", "NO", stEmpty, stEmpty, stEmpty\MaxTime:=10\BreakFlag:=errvar;
        TPWrite "CANCEL"\Num:=WAIT_MAX;
        IF command=1 THEN
        	poke_left;
        IF errvar=ERR_TP_MAXTIME OR command=2 main;
        ENDIF
         MAIN;
	ENDPROC
	PROC clap()
		MoveJ clap_home, v1500, z50, toolpen;
		Set doGrip;
        WaitTime .3;
		MoveJ clap_1, v1500, z50, toolpen;
        Reset doGrip;
        WaitTime .3;
        MoveJ clap_home, v1500, z50, toolpen;
        MoveJ clap_home, v1500, z50, toolpen;
		Set doGrip;
        WaitTime .3;
		MoveJ clap_1, v1500, z50, toolpen;
        Reset doGrip;
        WaitTime .3;
        MoveJ clap_home, v1500, z50, toolpen;
        MoveJ home, v1000, z50, toolpen;
        Set DO10_14;
		MoveJ yes_down, v1000, z50, toolpen;
		MoveJ yes_up, v1000, z50, toolpen;
        MoveJ yes_down, v1000, z50, toolpen;
		MoveJ yes_up, v1000, z50, toolpen;
        MoveJ yes_down, v1000, z50, toolpen;
		MoveJ yes_up, v1000, z50, toolpen;
        MoveJ home, v1000, z50, toolpen;
        MoveJ stare_left, v100, z50, toolpen;
	     RETURN;
	ENDPROC
	PROC rock_out()
        PLAY_MUSIC;
        Clear reg1;
        start_of_rock:
		MoveJ home, v1000, z50, toolpen;
      	MoveJ rockout, v500, z50, toolpen;
		MoveJ rockout10, v500, z50, toolpen;
		MoveJ rockout20, v500, z50, toolpen;
		MoveJ rockout30, v500, z50, toolpen;
		MoveJ rockout40, v500, z50, toolpen;
		Set DO10_14;
		MoveJ rockout50, v500, z50, toolpen;
		MoveJ rockout60, v200, z50, toolpen;
		MoveJ rockout70, v500, z50, toolpen;
		MoveL rockout80, v200, z50, toolpen;
		MoveL rockout90, v500, z50, toolpen;
		MoveJ rockout100, v200, z50, toolpen;
		MoveJ rockout110, v500, z50, toolpen;
		MoveJ rockout120, v200, z50, toolpen;
		MoveJ rockout130, v500, z50, toolpen;
		MoveJ rockout140, v200, z50, toolpen;
		MoveJ rockout150, v500, z50, toolpen;
		MoveJ rockout160, v200, z50, toolpen;
        MoveJ home, v1000, z50, toolpen;
		MoveJ rockout, v500, z50, toolpen;
		MoveJ rockout10, v500, z50, toolpen;
		MoveJ rockout20, v500, z50, toolpen;
		MoveJ rockout30, v500, z50, toolpen;
		MoveJ rockout40, v500, z50, toolpen;
		Set DO10_14;
		MoveJ rockout50, v500, z50, toolpen;
		MoveJ rockout60, v200, z50, toolpen;
		MoveJ rockout70, v500, z50, toolpen;
		MoveL rockout80, v200, z50, toolpen;
		MoveL rockout90, v500, z50, toolpen;
		MoveJ rockout100, v200, z50, toolpen;
		MoveJ rockout110, v500, z50, toolpen;
		MoveJ rockout120, v200, z50, toolpen;
		MoveJ rockout130, v500, z50, toolpen;
		MoveJ rockout140, v200, z50, toolpen;
		MoveJ rockout150, v500, z50, toolpen;
		MoveJ rockout160, v200, z50, toolpen;
        MoveJ home, v1000, z50, toolpen;
		MoveJ rockout, v500, z50, toolpen;
		MoveJ rockout10, v500, z50, toolpen;
		MoveJ rockout20, v500, z50, toolpen;
		MoveJ rockout30, v500, z50, toolpen;
		MoveJ rockout40, v500, z50, toolpen;
		Set DO10_14;
		MoveJ rockout50, v500, z50, toolpen;
		MoveJ rockout60, v200, z50, toolpen;
		MoveJ rockout70, v500, z50, toolpen;
		MoveL rockout80, v200, z50, toolpen;
		MoveL rockout90, v500, z50, toolpen;
		MoveJ rockout100, v200, z50, toolpen;
		MoveJ rockout110, v500, z50, toolpen;
		MoveJ rockout120, v200, z50, toolpen;
		MoveJ rockout130, v500, z50, toolpen;
		MoveJ rockout140, v200, z50, toolpen;
		MoveJ rockout150, v500, z50, toolpen;
		MoveJ rockout160, v200, z50, toolpen;
		MoveJ rockout170, v300, z50, toolpen;
		MoveJ rockout180, v300, z50, toolpen;
		MoveJ rockout190, v300, z50, toolpen;
		MoveJ rockout170, v300, z50, toolpen;
		MoveL rockout200, v300, z50, toolpen;
        !start of wiggle
		Set DO10_14;
		Set doGrip;
		Movej rockout210, v300, z1, toolpen;
		Movej rockout220, v300, z1, toolpen;
        Movej rockout210, v300, z1, toolpen;
		Movej rockout220, v300, z1, toolpen;
        Reset DO10_14;
        Reset doGrip;
        Movej rockout210, v300, z1, toolpen;
		Movej rockout220, v300, z1, toolpen;
        Set DO10_14;
        Movej rockout210, v300, z1, toolpen;
		Movej rockout220, v300, z1, toolpen;
        Movej rockout210, v300, z1, toolpen;
        Reset DO10_14;
		Movej rockout220, v300, z1, toolpen;
        Movej rockout210, v300, z1, toolpen;
		Movej rockout220, v300, z1, toolpen;
        !start of walk like a egyptian right
        MoveJ rockout260, v500, z1, toolpen;
        WaitTime 1;
        MoveJ rockout270, v500, z1, toolpen;
        WaitTime 1;
        MoveJ rockout260, v500, z1, toolpen;
        WaitTime 1;
         MoveJ rockout270, v500, z1, toolpen;
         WaitTime 1;
        MoveJ rockout260, v500, z1, toolpen;
        WaitTime 1;
        MoveJ rockout270, v500, z1, toolpen;
        WaitTime 1;
        MoveJ rockout260, v500, z1, toolpen;
        WaitTime 1;
        MoveJ home, v1000, z50, toolpen;
        !yes copy
        Set DO10_14;
		MoveJ yes_down, v1000, z50, toolpen;
		MoveJ yes_up, v1000, z50, toolpen;
        MoveJ yes_down, v1000, z50, toolpen;
		MoveJ yes_up, v1000, z50, toolpen;
        MoveJ yes_down, v1000, z50, toolpen;
		MoveJ yes_up, v1000, z50, toolpen;
        MoveJ home, v1000, z50, toolpen;
     !start of walk like a egyptian left
        MoveJ rockout280, v500, z50, toolpen;
        WaitTime 1;
        MoveJ rockout290, v500, z50, toolpen;
        WaitTime 1;
        MoveJ rockout280, v500, z50, toolpen;
        WaitTime 1;
        MoveJ rockout290, v500, z50, toolpen;
        WaitTime 1;
        MoveJ rockout280, v500, z50, toolpen;
        WaitTime 1;
        MoveJ rockout290, v500, z50, toolpen;
        WaitTime 1;
        MoveJ rockout280, v500, z50, toolpen;
        Incr reg1;
    IF reg1=2 THEN PLAY_MUSIC;
    ELSE GOTO start_of_rock;
    ENDIF
     MAIN;
   	ENDPROC
	PROC photo_activate()
	WaitUntil DI10_9=1;
    MoveJ look_left_home30, v100, fine, toolpen;
    MoveJ look_left_home40, v100, fine, toolpen;
	MoveJ POKE, v1000, fine, toolpen;
    Set doGrip;
    MoveJ look_left_home40, v1000, z50, toolpen;
    clap;
	ENDPROC
	PROC poke_left()
	 WaitUntil DI10_9=1;
     WaitTime 2;
	MoveJ POKE, v1000, fine, toolpen;
    Set doGrip;
     MoveJ look_left_home40, v1000, z50, toolpen;
    clap;
	ENDPROC
    PROC PONG_DOINK()
    MoveJ home, v1000, z50, toolpen;
    MoveJ doink_pickup1, v500, z50, toolsuck\WObj:=wobjgraph;
    MoveL doink_pickup10, v1000, fine, toolsuck\WObj:=wobjgraph;
    Set doVacume;
    MoveL doink_pickup1, v1000, z50, toolsuck\WObj:=wobjgraph;
    MoveJ doink_pickup51, v500, z50, toolsuck\WObj:=wobjgraph;
    MoveJ doink_pickup11, v500, z50, toolsuck\WObj:=wobjgraph;
    MoveC doink_pickup81, doink_pickup91, v3000, z200, toolsuck\WObj:=wobjgraph;
    WaitTime 0.5;
    Reset doVacume;
    clap;
    ENDPROC
     PROC BALL_MADNESS()
    Clear reg1;
    TPReadNum reg2, "ENTER TIMES TO THROW 1-10. ONCE PHOTOEYE IS MADE BALL MADNESS BEGINS";
    WaitUntil DI10_9=1;
    start_of_doink:
    MoveJ home, v1000, z50, toolpen;
    MoveJ doink_pickup1, v500, z50, toolsuck\WObj:=wobjgraph;
    MoveL doink_pickup10, v1000, fine, toolsuck\WObj:=wobjgraph;
    Set doVacume;
    MoveL doink_pickup1, v1000, z50, toolsuck\WObj:=wobjgraph;
    MoveJ doink_pickup51, v500, z50, toolsuck\WObj:=wobjgraph;
    MoveJ doink_pickup11, v500, z50, toolsuck\WObj:=wobjgraph;
    MoveC doink_pickup81, doink_pickup91, v3000, z200, toolsuck\WObj:=wobjgraph;
    WaitTime 0.5;
    Reset doVacume;
     Incr reg1;
     MoveJ doink_pickup51, v500, z50, toolsuck\WObj:=wobjgraph;
    IF reg1=reg2 THEN YES;
    ELSE GOTO start_of_doink;
    ENDIF
         RETURN;
    ENDPROC

    PROC SCRATCH1()
!!!!!!!!!!!Idle code
     MoveJ scratch, v200, z50, toolpen;
    Set doGrip;
     Set DO10_14;
  MoveJ scratch10, v500, z50, toolpen;
   MoveJ scratch20, V500, z50, toolpen;
     WaitTime .5;
    MoveJ scratch10, v500, z50, toolpen;
   MoveJ scratch20, V500, z50, toolpen;
     WaitTime .5;
     MoveJ scratch10, v500, z50, toolpen;
    MoveJ scratch20, V500, z50, toolpen;
   WaitTime .5;
    RESET DO10_14;
     MoveJ scratch30, v200, z50, toolpen;
    MoveJ stare_left, v300, z150, toolpen;
     RETURN;
         ENDPROC
    PROC COCK_HEAD ()
     MoveJ stare_left, v300, z150, toolpen;

!!!!!!!!!!!Idle code
MoveJ stare_left10, v300, z150, toolpen;
WaitTime 1;
MoveJ stare_left20, v300, z150, toolpen;

!!!!!!!!!!!Idle code

      ENDPROC
     PROC LICK ()
     MoveJ stare_left, v300, z150, toolpen;

!!!!!!!!!!!Idle code
MoveJ stare_left30, v300, fine, toolpen;
Set DO10_14;
WaitTime 0.7;
MoveJ lick1, v100, z10, toolpen;
MoveJ lick11, v100, z10, toolpen;
Reset DO10_14;

!!!!!!!!!!!Idle code

       RETURN;
        ENDPROC
        PROC PLAY_MUSIC ()
     MoveJ stare_left, v300, z150, toolpen;
      MoveJ above_play, v100, z10, toolpen;
MoveL press_play, v100, fine, toolpen;
WaitTime 0.3;
Reset DO10_14;
 MoveJ stare_left, v300, z150, toolpen;

       RETURN;
        ENDPROC
     PROC LOOK_ABOUT ()
       MoveJ stare_left, v300, z150, toolpen;

!!!!!!!!!!!Idle code
MoveJ look_at_feeder, v300, z150, toolpen;
WaitTime 0.7;
MoveJ look_at_feeder10, v150, z150, toolpen;
WaitTime 2;
MoveJ look_at_feeder20, v150, z150, toolpen;
Set DO10_14;
ConfL \Off;
MoveL look_at_feeder50, v150, z150, toolpen;
MoveL look_at_feeder30, v300, z150, toolpen;
MoveL look_at_feeder40, v300, z150, toolpen;
MoveL look_at_feeder30, v300, z150, toolpen;
Reset DO10_14;
ConfL \on;
!!!!!!!!!!!Idle code

       RETURN;
        ENDPROC
       PROC LOOK_UP_DN ()

!!!!!!!!!!!Idle code
MoveJ look_up_dn1, v300, z150, toolpen;
MoveJ look_up_dn11, v300, z150, toolpen;
MoveJ look_up_dn21, v300, z150, toolpen;
MoveJ look_up_dn31, v300, z150, toolpen;
MoveJ look_up_dn41, v300, z150, toolpen;
MoveJ look_up_dn51, v300, z150, toolpen;

!!!!!!!!!!!Idle code
 MAIN;
        ENDPROC
         PROC DEMO ()
              TPReadNum reg2, "ENTER SECONDS BETWEEN EACH CYCLE";
         DEMOCYCLE:
!!!!!!!!!!!CLAP
WaitTime reg2;
MoveJ clap_home, v1500, z50, toolpen;
		Set doGrip;
        WaitTime .3;
		MoveJ clap_1, v1500, z50, toolpen;
        Reset doGrip;
        WaitTime .3;
        MoveJ clap_home, v1500, z50, toolpen;
        MoveJ clap_home, v1500, z50, toolpen;
		Set doGrip;
        WaitTime .3;
		MoveJ clap_1, v1500, z50, toolpen;
        Reset doGrip;
        WaitTime .3;
        MoveJ clap_home, v1500, z50, toolpen;
        MoveJ home, v1000, z50, toolpen;
        Set DO10_14;
		MoveJ yes_down, v1000, z50, toolpen;
		MoveJ yes_up, v1000, z50, toolpen;
        MoveJ yes_down, v1000, z50, toolpen;
		MoveJ yes_up, v1000, z50, toolpen;
        MoveJ yes_down, v1000, z50, toolpen;
		MoveJ yes_up, v1000, z50, toolpen;
        MoveJ home, v1000, z50, toolpen;
        MoveJ stare_left, v100, z50, toolpen;
        !!!!!!!!!!!COCK_HEAD
  WaitTime reg2;
        MoveJ stare_left, v300, z150, toolpen;
MoveJ stare_left10, v300, z150, toolpen;
WaitTime 1;
MoveJ stare_left20, v300, z150, toolpen;
        !!!!!!!!!!!LICK
MoveJ stare_left, v300, z150, toolpen;
MoveJ stare_left30, v300, fine, toolpen;
Set DO10_14;
WaitTime 0.7;
MoveJ lick1, v100, z10, toolpen;
MoveJ lick11, v100, z10, toolpen;
Reset DO10_14;
     WaitTime reg2;
        !!!!!!!!!!!LOOK_ABOUT
           MoveJ stare_left, v300, z150, toolpen;
MoveJ look_at_feeder, v300, z150, toolpen;
WaitTime 0.7;
MoveJ look_at_feeder10, v150, z150, toolpen;
WaitTime 2;
MoveJ look_at_feeder20, v150, z150, toolpen;
Set DO10_14;
ConfL \Off;
MoveL look_at_feeder50, v150, z150, toolpen;
MoveL look_at_feeder30, v300, z150, toolpen;
MoveL look_at_feeder40, v300, z150, toolpen;
MoveL look_at_feeder30, v300, z150, toolpen;
Reset DO10_14;
ConfL \on;
       WaitTime reg2;
        !!!!!!!!!!!LOOK_LEFT
        MoveJ look_left_home, v500, z50, toolpen;
		MoveJ look_left_home10, v100, fine, toolpen;
        Set doGrip;
        WaitTime .5;
        Reset doGrip;
        WaitTime .5;
		MoveJ look_left_home20, v100, fine, toolpen;
         Set doGrip;
        WaitTime .5;
        Reset doGrip;
        WaitTime .5;
        Set DO10_14;
        WaitTime 1;
        Reset DO10_14;
        WaitTime 1;
        MoveJ look_left_home30, v100, fine, toolpen;
        MoveJ look_left_home40, v100, fine, toolpen;
     WaitTime reg2;
        !!!!!!!!!!!LOOK_UP_DN
        MoveJ look_up_dn1, v300, z150, toolpen;
MoveJ look_up_dn11, v300, z150, toolpen;
MoveJ look_up_dn21, v300, z150, toolpen;
MoveJ look_up_dn31, v300, z150, toolpen;
MoveJ look_up_dn41, v300, z150, toolpen;
MoveJ look_up_dn51, v300, z150, toolpen;
     WaitTime reg2;
        !!!!!!!!!!!NO
       MoveJ home, v1000, z50, toolpen;
        Set DO10_14;
		MoveJ no_left, v1000, z50, toolpen;
		MoveJ no_right, v1000, z50, toolpen;
        MoveJ no_left, v1000, z50, toolpen;
		MoveJ no_right, v1000, z50, toolpen;
        MoveJ no_left, v1000, z50, toolpen;
		MoveJ no_right, v1000, z50, toolpen;
        MoveJ home, v1000, z50, toolpen;
      WaitTime reg2;
        !!!!!!!!!!!SCRATCH1
          MoveJ scratch, v200, z50, toolpen;
    Set doGrip;
     Set DO10_14;
  MoveJ scratch10, v500, z50, toolpen;
   MoveJ scratch20, V500, z50, toolpen;
     WaitTime .5;
    MoveJ scratch10, v500, z50, toolpen;
   MoveJ scratch20, V500, z50, toolpen;
     WaitTime .5;
     MoveJ scratch10, v500, z50, toolpen;
    MoveJ scratch20, V500, z50, toolpen;
   WaitTime .5;
    RESET DO10_14;
     MoveJ scratch30, v200, z50, toolpen;
    MoveJ stare_left, v300, z150, toolpen;
       WaitTime reg2;
        !!!!!!!!!!!YES
        MoveJ home, v1000, z50, toolpen;
        Set DO10_14;
		MoveJ yes_down, v1000, z50, toolpen;
		MoveJ yes_up, v1000, z50, toolpen;
        MoveJ yes_down, v1000, z50, toolpen;
		MoveJ yes_up, v1000, z50, toolpen;
        MoveJ yes_down, v1000, z50, toolpen;
		MoveJ yes_up, v1000, z50, toolpen;
        MoveJ home, v1000, z50, toolpen;
    WaitTime reg2;
         !!!!!!!!!!!Rockout
          start_of_rock:
		MoveJ home, v1000, z50, toolpen;
		MoveJ rockout, v500, z50, toolpen;
		MoveJ rockout10, v500, z50, toolpen;
		MoveJ rockout20, v500, z50, toolpen;
		MoveJ rockout30, v500, z50, toolpen;
		MoveJ rockout40, v500, z50, toolpen;
		Set DO10_14;
		MoveJ rockout50, v500, z50, toolpen;
		MoveJ rockout60, v200, z50, toolpen;
		MoveJ rockout70, v500, z50, toolpen;
		MoveL rockout80, v200, z50, toolpen;
		MoveL rockout90, v500, z50, toolpen;
		MoveJ rockout100, v200, z50, toolpen;
		MoveJ rockout110, v500, z50, toolpen;
		MoveJ rockout120, v200, z50, toolpen;
		MoveJ rockout130, v500, z50, toolpen;
		MoveJ rockout140, v200, z50, toolpen;
		MoveJ rockout150, v500, z50, toolpen;
		MoveJ rockout160, v200, z50, toolpen;
        MoveJ home, v1000, z50, toolpen;
		MoveJ rockout, v500, z50, toolpen;
		MoveJ rockout10, v500, z50, toolpen;
		MoveJ rockout20, v500, z50, toolpen;
		MoveJ rockout30, v500, z50, toolpen;
		MoveJ rockout40, v500, z50, toolpen;
		Set DO10_14;
		MoveJ rockout50, v500, z50, toolpen;
		MoveJ rockout60, v200, z50, toolpen;
		MoveJ rockout70, v500, z50, toolpen;
		MoveL rockout80, v200, z50, toolpen;
		MoveL rockout90, v500, z50, toolpen;
		MoveJ rockout100, v200, z50, toolpen;
		MoveJ rockout110, v500, z50, toolpen;
		MoveJ rockout120, v200, z50, toolpen;
		MoveJ rockout130, v500, z50, toolpen;
		MoveJ rockout140, v200, z50, toolpen;
		MoveJ rockout150, v500, z50, toolpen;
		MoveJ rockout160, v200, z50, toolpen;
        MoveJ home, v1000, z50, toolpen;
		MoveJ rockout, v500, z50, toolpen;
		MoveJ rockout10, v500, z50, toolpen;
		MoveJ rockout20, v500, z50, toolpen;
		MoveJ rockout30, v500, z50, toolpen;
		MoveJ rockout40, v500, z50, toolpen;
		Set DO10_14;
		MoveJ rockout50, v500, z50, toolpen;
		MoveJ rockout60, v200, z50, toolpen;
		MoveJ rockout70, v500, z50, toolpen;
		MoveL rockout80, v200, z50, toolpen;
		MoveL rockout90, v500, z50, toolpen;
		MoveJ rockout100, v200, z50, toolpen;
		MoveJ rockout110, v500, z50, toolpen;
		MoveJ rockout120, v200, z50, toolpen;
		MoveJ rockout130, v500, z50, toolpen;
		MoveJ rockout140, v200, z50, toolpen;
		MoveJ rockout150, v500, z50, toolpen;
		MoveJ rockout160, v200, z50, toolpen;
		MoveJ rockout170, v300, z50, toolpen;
		MoveJ rockout180, v300, z50, toolpen;
		MoveJ rockout190, v300, z50, toolpen;
		MoveJ rockout170, v300, z50, toolpen;
		MoveL rockout200, v300, z50, toolpen;
        !start of wiggle
		Set DO10_14;
		Set doGrip;
		Movej rockout210, v300, z1, toolpen;
		Movej rockout220, v300, z1, toolpen;
        Movej rockout210, v300, z1, toolpen;
		Movej rockout220, v300, z1, toolpen;
        Reset DO10_14;
        Reset doGrip;
        Movej rockout210, v300, z1, toolpen;
		Movej rockout220, v300, z1, toolpen;
        Set DO10_14;
        Movej rockout210, v300, z1, toolpen;
		Movej rockout220, v300, z1, toolpen;
        Movej rockout210, v300, z1, toolpen;
        Reset DO10_14;
		Movej rockout220, v300, z1, toolpen;
        Movej rockout210, v300, z1, toolpen;
		Movej rockout220, v300, z1, toolpen;
        !start of walk like a egyptian right
        MoveJ rockout260, v500, z1, toolpen;
        WaitTime 1;
        MoveJ rockout270, v500, z1, toolpen;
        WaitTime 1;
        MoveJ rockout260, v500, z1, toolpen;
        WaitTime 1;
         MoveJ rockout270, v500, z1, toolpen;
         WaitTime 1;
        MoveJ rockout260, v500, z1, toolpen;
        WaitTime 1;
        MoveJ rockout270, v500, z1, toolpen;
        WaitTime 1;
        MoveJ rockout260, v500, z1, toolpen;
        WaitTime 1;
        MoveJ home, v1000, z50, toolpen;
        !yes copy
        Set DO10_14;
		MoveJ yes_down, v1000, z50, toolpen;
		MoveJ yes_up, v1000, z50, toolpen;
        MoveJ yes_down, v1000, z50, toolpen;
		MoveJ yes_up, v1000, z50, toolpen;
        MoveJ yes_down, v1000, z50, toolpen;
		MoveJ yes_up, v1000, z50, toolpen;
        MoveJ home, v1000, z50, toolpen;
     !start of walk like a egyptian left
        MoveJ rockout280, v500, z50, toolpen;
        WaitTime 1;
        MoveJ rockout290, v500, z50, toolpen;
        WaitTime 1;
        MoveJ rockout280, v500, z50, toolpen;
        WaitTime 1;
        MoveJ rockout290, v500, z50, toolpen;
        WaitTime 1;
        MoveJ rockout280, v500, z50, toolpen;
        WaitTime 1;
        MoveJ rockout290, v500, z50, toolpen;
        WaitTime 1;
        MoveJ rockout280, v500, z50, toolpen;
           GOTO DEMOCYCLE;
        ENDPROC
        PROC CupDrop()
        CUPJUMP:
        reg5:=0;
        TPErase;
        TPwrite "MOVE HAND IN FRONT OF YELLOW SENSOR TO       DROP THE BALL INTO THE CUP";
        !Pick up Ball then move to Home
        IWatch drop;
        MoveJ home, v1000, z50, toolpen;
        MoveJ doink_pickup1, v500, z50, toolsuck\WObj:=wobjgraph;
        MoveL doink_pickup10, v1000, fine, toolsuck\WObj:=wobjgraph;
        Set doVacume;
        MoveJ cupdrop1, v500, z50, toolsuck\WObj:=wobjgraph;
             WHILE TRUE DO
            !runs circle loop until reg5 set to zero in vacdropnow trap
                IF reg5=0 THEN
              MoveAbsJ jpos20\NoEOffs, v300, z200, toolsuck\WObj:=wobjgraph;
              MoveAbsJ jpos30\NoEOffs, v300, z200, toolsuck\WObj:=wobjgraph;
                    ELSE
                    GOTO cupjump1;
             ENDIF
        ENDWHILE
        cupjump1:
        TPReadFK command, "TRY AGAIN", "YES", "NO", stEmpty, stEmpty, stEmpty\MaxTime:=10\BreakFlag:=errvar;
        TPWrite "CANCEL"\Num:=WAIT_MAX;
        IF command=1 THEN
        	GOTO CUPJUMP;
        IF command=2 main;
        ENDIF
        main;
          ENDPROC
        TRAP VacDropNow
		Reset doVacume;
        reg5:=1;
	ENDTRAP
	PROC setup_red()
		TPWrite "HOW LONG DOES IT TAKE?";
        WaitTime 2;
        TPWrite "HOW CAN WE MAKE IT BETTER?";
         WaitTime 2;
        TPWrite "SINGLE MINUTE EXCHANGE OF DIE";
         WaitTime 2;
        TPWrite "SETUP REDUCTION IS COMMON SENSE ";
         WaitTime 2;
        TPWrite "COMMON SENSE IS VERY UNCOMMON";
         WaitTime 2;
         TPWrite "DON'T DO IT GOOFY'S WAY! ";
         WaitTime 1;
        TPWrite "ENROLL IN SETUP REDUCTION CLASS TODAY!";
        ClkReset clock1;
        ClkSTART clock1;
        TPWrite "CYCLE TIME="\Num:=ClkRead(clock1);
        MoveJ setuphome, v100, z50, toolsuck\WObj:=setup;
        TPShow TP_LATEST;
		!picup seat at load 1
        MoveJ setup_aboveseat_load1, v100, z50, toolsuck\WObj:=setup;
        Set doVacume;
		MoveL setup_atseat_load1, v50, fine, toolsuck\WObj:=setup;
		WaitTime 1;
		MoveL setup_aboveseat_load1, v100, fine, toolsuck\WObj:=setup;
		!place seat on frame
        MoveL setup_aboveframe, v100, fine, toolsuck\WObj:=setup;
		MoveL setup_place_seat_on_frame, v100, fine, toolsuck\WObj:=setup;
		Reset doVacume;
		WaitTime 1;
        MoveL setup_aboveframe, v100, fine, toolsuck\WObj:=setup;

		!pickup body load 2

        MoveJ setup_abovebody_load2, v100, fine, toolsuck\WObj:=setup;
        Set doVacume;
		MoveL setup_atbody_load2, v100, fine, toolsuck\WObj:=setup;
		WaitTime 1;
		MoveL setup_abovebody_load2, v100, fine, toolsuck\WObj:=setup;
        !place body on frame
        MoveL setup_body_above_frame, v100, fine, toolsuck\WObj:=setup;
		MoveL setup_place_body_on_frame, v100, fine, toolsuck\WObj:=setup;
		Reset doVacume;
		WaitTime 1;
		MoveL setup_body_above_frame, v100, fine, toolsuck\WObj:=setup;
         !glue car
		MoveJ setup_above_pen, v200, z50, toolpen\WObj:=setup;
        Movel setup_at_pen, v200, fine, toolpen\WObj:=setup;
        Set doGrip;
        WaitTime 0.5;
        Movel setup_above_pen, v200, fine, toolpen\WObj:=setup;
        MoveJ setup_pen_above_frame, v400, z50, toolpen\WObj:=setup;
        !start of reorient wasted move
        MoveJ setup_pen_glue1_frame, v10, z50, toolpen\WObj:=setup;
        MoveJ setup_pen_glue2_frame, v10, z50, toolpen\WObj:=setup;
        MoveJ setup_pen_glue3_frame, v10, z50, toolpen\WObj:=setup;
        MoveJ setup_pen_glue4_frame, v10, z50, toolpen\WObj:=setup;
        MoveJ setup_pen_above_frame, v10, z50, toolpen\WObj:=setup;
        !start of glue seq
        MoveJ setup_pen_glue5_frame, v100, z50, toolpen\WObj:=setup;
        MoveJ setup_pen_glue6_frame, v100, z50, toolpen\WObj:=setup;
        MoveJ setup_pen_glue7_frame, v100, z50, toolpen\WObj:=setup;
        MoveJ setup_pen_glue8_frame, v100, z50, toolpen\WObj:=setup;
        MoveJ setup_pen_above_frame, v400, z50, toolpen\WObj:=setup;
        MoveJ setup_above_pen, v400, z50, toolpen\WObj:=setup;
         Movel setup_at_pen, v200, fine, toolpen\WObj:=setup;
         WaitTime 0.5;
         Reset doGrip;
         Movel setup_above_pen, v200, fine, toolpen\WObj:=setup;
        !pick body off of frame
        MoveL setup_body_above_frame, v100, fine, toolsuck\WObj:=setup;
		MoveL setup_place_body_on_frame, v100, fine, toolsuck\WObj:=setup;
        set doVacume;
		WaitTime 1;
		MoveL setup_body_above_frame, v100, fine, toolsuck\WObj:=setup;
        !put body at load 2
        MoveJ setup_abovebody_load2, v100, fine, toolsuck\WObj:=setup;
		MoveL setup_atbody_load2, v100, fine, toolsuck\WObj:=setup;
        Reset doVacume;
		WaitTime 1;
		MoveL setup_abovebody_load2, v100, fine, toolsuck\WObj:=setup;
        !pick seat off of frame
        MoveL setup_aboveframe, v100, fine, toolsuck\WObj:=setup;
		MoveL setup_place_seat_on_frame, v100, fine, toolsuck\WObj:=setup;
        set doVacume;
		WaitTime 1;
		MoveL setup_aboveframe, v100, fine, toolsuck\WObj:=setup;
        !put seat at load 1
         MoveJ setup_aboveseat_load1, v100, z50, toolsuck\WObj:=setup;
		MoveL setup_atseat_load1, v50, fine, toolsuck\WObj:=setup;
        Reset doVacume;
		WaitTime 1;
		MoveL setup_aboveseat_load1, v100, fine, toolsuck\WObj:=setup;
         TPWrite "CYCLE TIME="\Num:=ClkRead(clock1);
         WaitTime 5;
         setup_red;

	ENDPROC
ENDMODULE

--- Backups/120-501447/HOME/lab7/MainModule.mod ---
MODULE MainModule
	TASK PERS tooldata tPen:=[TRUE,[[0.147757,-83.6911,144.451],[0.738156,0.674482,-0.0103991,-0.00950206]],[0.8,[1.7,0,108.7],[1,0,0,0],0.011,0.006,0.009]];
	CONST robtarget p30:=[[469.22,99.75,8.79],[0.0216335,0.64282,0.765703,-0.00355185],[0,0,0,1],[9E+09,9E+09,9E+09,9E+09,9E+09,9E+09]];
	CONST robtarget pstart:=[[512.08,-48.21,10.23],[0.0215519,0.642623,0.765869,-0.00379738],[-1,-1,0,1],[9E+09,9E+09,9E+09,9E+09,9E+09,9E+09]];
	CONST robtarget p10:=[[268.52,32.55,142.20],[0.0387242,0.836099,0.54718,0.00566096],[0,0,0,1],[9E+09,9E+09,9E+09,9E+09,9E+09,9E+09]];
	CONST robtarget p20:=[[268.52,32.55,29.70],[0.0387219,0.8361,0.547177,0.00566567],[0,0,0,1],[9E+09,9E+09,9E+09,9E+09,9E+09,9E+09]];
	CONST robtarget p40:=[[505.98,113.33,4.46],[0.0367854,0.831559,0.554195,0.00482753],[0,0,0,1],[9E+09,9E+09,9E+09,9E+09,9E+09,9E+09]];
	CONST robtarget p50:=[[461.62,115.15,-8.30],[0.0367965,0.831555,0.5542,0.00481934],[0,0,0,1],[9E+09,9E+09,9E+09,9E+09,9E+09,9E+09]];
	CONST robtarget p60:=[[525.97,169.03,3.52],[0.0368121,0.8315,0.554282,0.00472824],[0,0,0,1],[9E+09,9E+09,9E+09,9E+09,9E+09,9E+09]];
	CONST robtarget p70:=[[597.29,115.27,0.65],[0.0368322,0.831492,0.554294,0.00471092],[0,0,0,1],[9E+09,9E+09,9E+09,9E+09,9E+09,9E+09]];
	CONST robtarget p80:=[[569.04,115.26,0.68],[0.036874,0.831516,0.554254,0.00474228],[0,0,0,1],[9E+09,9E+09,9E+09,9E+09,9E+09,9E+09]];
	CONST robtarget p90:=[[579.87,-35.31,-1.57],[0.0368611,0.831471,0.554322,0.00471824],[0,0,0,1],[9E+09,9E+09,9E+09,9E+09,9E+09,9E+09]];
	CONST robtarget p100:=[[547.53,-9.26,-1.58],[0.0368624,0.831474,0.554318,0.00469294],[0,0,0,1],[9E+09,9E+09,9E+09,9E+09,9E+09,9E+09]];
	CONST robtarget p110:=[[532.30,-194.48,243.92],[0.0367212,0.831611,0.55412,0.00498134],[-1,0,0,1],[9E+09,9E+09,9E+09,9E+09,9E+09,9E+09]];
	TASK PERS wobjdata wFixture1:=[FALSE,TRUE,"",[[0,0,0],[1,0,0,0]],[[357.689,-176.134,-17.7192],[0.999991,-0.00111829,0.000705852,-0.00392021]]];
	TASK PERS wobjdata wobj1:=[FALSE,TRUE,"",[[0,0,0],[1,0,0,0]],[[372.049,-59.0817,-2.31291],[0.999964,0.00101619,0.00195787,0.00815211]]];
	PROC main()
		MoveJ p10, v1000, z50, tPen\WObj:=wobj1;
		MoveL p20, v1000, fine, tPen\WObj:=wobj1;
		Set doGrip;
		MoveL p10, v1000, fine, tPen\WObj:=wobj1;
		MoveL [[523.80,-56.63,-8.74],[0.0367413,0.831596,0.554142,0.00493633],[0,0,0,1],[9E+09,9E+09,9E+09,9E+09,9E+09,9E+09]], v1000, fine, tPen\WObj:=wobj1;
		MoveL [[449.04,-57.95,-7.57],[0.0367587,0.831587,0.554155,0.00488328],[0,0,1,1],[9E+09,9E+09,9E+09,9E+09,9E+09,9E+09]], v1000, fine, tPen\WObj:=wobj1;
		MoveL [[497.17,94.80,-7.58],[0.0367718,0.831577,0.554169,0.00486949],[0,0,0,1],[9E+09,9E+09,9E+09,9E+09,9E+09,9E+09]], v1000, fine, tPen\WObj:=wobj1;
		MoveL [[524.39,-59.04,-6.34],[0.037286,0.83168,0.553975,0.00527583],[0,0,0,1],[9E+09,9E+09,9E+09,9E+09,9E+09,9E+09]], v1000, fine, tPen\WObj:=wobj1;
		MoveL p10, v1000, fine, tPen;
		MoveL p20, v1000, fine, tPen;
		Reset doGrip;
	ENDPROC
	PROC rGotoCal()
		MoveAbsJ jposCal\NoEOffs, v1000, z50, tPen\WObj:=wobj1;
	ENDPROC
ENDMODULE

--- Backups/120-501447/HOME/Trangle/MainModule.mod ---
MODULE MainModule
	TASK PERS tooldata tPen:=[TRUE,[[0.147757,-83.6911,144.451],[0.738156,0.674482,-0.0103991,-0.00950206]],[0.8,[1.7,0,108.7],[1,0,0,0],0.011,0.006,0.009]];
	CONST robtarget p30:=[[469.22,99.75,8.79],[0.0216335,0.64282,0.765703,-0.00355185],[0,0,0,1],[9E+09,9E+09,9E+09,9E+09,9E+09,9E+09]];
	CONST robtarget pstart:=[[512.08,-48.21,10.23],[0.0215519,0.642623,0.765869,-0.00379738],[-1,-1,0,1],[9E+09,9E+09,9E+09,9E+09,9E+09,9E+09]];
	CONST robtarget p10:=[[532.31,-194.48,243.93],[0.0367381,0.831611,0.554119,0.00499251],[-1,0,0,1],[9E+09,9E+09,9E+09,9E+09,9E+09,9E+09]];
	CONST robtarget p20:=[[520.51,-195.94,22.35],[0.0374863,0.834786,0.549146,-0.0128487],[-1,0,0,1],[9E+09,9E+09,9E+09,9E+09,9E+09,9E+09]];
	CONST robtarget p40:=[[505.98,113.33,4.46],[0.0367854,0.831559,0.554195,0.00482753],[0,0,0,1],[9E+09,9E+09,9E+09,9E+09,9E+09,9E+09]];
	CONST robtarget p50:=[[461.62,115.15,-8.30],[0.0367965,0.831555,0.5542,0.00481934],[0,0,0,1],[9E+09,9E+09,9E+09,9E+09,9E+09,9E+09]];
	CONST robtarget p60:=[[525.97,169.03,3.52],[0.0368121,0.8315,0.554282,0.00472824],[0,0,0,1],[9E+09,9E+09,9E+09,9E+09,9E+09,9E+09]];
	CONST robtarget p70:=[[597.29,115.27,0.65],[0.0368322,0.831492,0.554294,0.00471092],[0,0,0,1],[9E+09,9E+09,9E+09,9E+09,9E+09,9E+09]];
	CONST robtarget p80:=[[569.04,115.26,0.68],[0.036874,0.831516,0.554254,0.00474228],[0,0,0,1],[9E+09,9E+09,9E+09,9E+09,9E+09,9E+09]];
	CONST robtarget p90:=[[579.87,-35.31,-1.57],[0.0368611,0.831471,0.554322,0.00471824],[0,0,0,1],[9E+09,9E+09,9E+09,9E+09,9E+09,9E+09]];
	CONST robtarget p100:=[[547.53,-9.26,-1.58],[0.0368624,0.831474,0.554318,0.00469294],[0,0,0,1],[9E+09,9E+09,9E+09,9E+09,9E+09,9E+09]];
	CONST robtarget p110:=[[532.30,-194.48,243.92],[0.0367212,0.831611,0.55412,0.00498134],[-1,0,0,1],[9E+09,9E+09,9E+09,9E+09,9E+09,9E+09]];
	TASK PERS wobjdata wFixture1:=[FALSE,TRUE,"",[[0,0,0],[1,0,0,0]],[[357.689,-176.134,-17.7192],[0.999991,-0.00111829,0.000705852,-0.00392021]]];
	TASK PERS wobjdata wobj1:=[FALSE,TRUE,"",[[0,0,0],[1,0,0,0]],[[372.049,-59.0817,-2.31291],[0.999964,0.00101619,0.00195787,0.00815211]]];
	PROC main()
		MoveJ p10, v1000, z50, tPen\WObj:=wobj1;
		MoveL p20, v1000, fine, tPen\WObj:=wobj1;
		Set doGrip;
		MoveL p10, v1000, fine, tPen;
		MoveL [[523.80,-56.63,-8.74],[0.0367413,0.831596,0.554142,0.00493633],[0,0,0,1],[9E+09,9E+09,9E+09,9E+09,9E+09,9E+09]], v1000, fine, tPen;
		MoveL [[449.04,-57.95,-7.57],[0.0367587,0.831587,0.554155,0.00488328],[0,0,1,1],[9E+09,9E+09,9E+09,9E+09,9E+09,9E+09]], v1000, fine, tPen;
		MoveL [[497.17,94.80,-7.58],[0.0367718,0.831577,0.554169,0.00486949],[0,0,0,1],[9E+09,9E+09,9E+09,9E+09,9E+09,9E+09]], v1000, fine, tPen;
		MoveL [[524.39,-59.04,-6.34],[0.037286,0.83168,0.553975,0.00527583],[0,0,0,1],[9E+09,9E+09,9E+09,9E+09,9E+09,9E+09]], v1000, fine, tPen;
		MoveL p10, v1000, fine, tPen;
		MoveL p20, v1000, fine, tPen;
		Reset doGrip;
	ENDPROC
ENDMODULE

--- Backups/120-501447/HOME/Trangle/Wobj_wFixture1.mod ---
MODULE Wobj_wFixture1
	! Points are read in order of declaration.
  ! Please do not change the order of points!

